// TIA Portal project "RHIKOR Barranquill Agua Renovada_V19" (V19)

(* hardware
DEVICE "S7-1500/ET200MP station_1"  S7-1500 station
   slot 0: "Rail_0"  Rack  6ES7 590-1***0-0AA0
   slot 1: "6ES7 511-1AL03-0AB0"  CPU 1511-1 PN  6ES7 511-1AL03-0AB0  V3.0
      slot 3: "CPU display_1"  6ES7591-1AA00-0AA0
      slot 32768: "PROFINET interface_1"  X1
         slot 32769: "Port_1"  X1 P1
         slot 32770: "Port_2"  X1 P2
      slot 34817: "Virtual CP interface port_1"  Virtual CP interface port  Virtual CP interface port
   slot 2: "PS 25W 24VDC_1"  PS 25W 24VDC  6ES7 505-0KA00-0AB0  V1.1
DEVICE "HMI_1"  KTP900 Basic PN
   slot 0: "HMI_1"  KTP900 Basic PN  6AV2 123-2JB03-0AX0  17.0.0.0
   slot 1: "HMI_RT_1"  KTP900 Basic PN  6AV2 123-2JB03-0AX0  17.0.0.0
   slot 5: "HMI_1.IE_CP_1"  PROFINET Interface  17.0.0.0
      slot 1: "hmixb110d0"  PROFINET Interface
         slot 1: "Port_1"  Port
DEVICE "SCALANCE X005"  SCALANCE X-Station
   slot 0: "SCALANCE X rack"  Rail
   slot 0: "Switch_1"  6GK5 005-0BA00-1AB2  V1.0
DEVICE "ET 200SP station_1"  ET 200SP-Station
   slot 0: "Rack_0"  Rack  6ES5 710-8MAx1
   slot 0: "et200sp"  IM 155-6 PN ST  6ES7 155-6AU02-0BN0  V6.1
   slot 1: "DI 16x24VDC ST_1"  DI 16x24VDC ST  6ES7 131-6BH01-0BA0  V0.0
      slot 1: "DI 16x24VDC ST_1"  DI 16x24VDC ST
   slot 2: "DI 16x24VDC ST_2"  DI 16x24VDC ST  6ES7 131-6BH01-0BA0  V0.0
      slot 1: "DI 16x24VDC ST_2"  DI 16x24VDC ST
   slot 3: "DI 16x24VDC ST_3"  DI 16x24VDC ST  6ES7 131-6BH01-0BA0  V0.0
      slot 1: "DI 16x24VDC ST_3"  DI 16x24VDC ST
   slot 4: "DI 16x24VDC ST_4"  DI 16x24VDC ST  6ES7 131-6BH01-0BA0  V0.0
      slot 1: "DI 16x24VDC ST_4"  DI 16x24VDC ST
   slot 5: "DQ 16x24VDC/0.5A ST_1"  DQ 16x24VDC/0.5A ST  6ES7 132-6BH01-0BA0  V0.0
      slot 1: "DQ 16x24VDC/0.5A ST_1"  DQ 16x24VDC/0.5A ST
   slot 6: "DQ 16x24VDC/0.5A ST_2"  DQ 16x24VDC/0.5A ST  6ES7 132-6BH01-0BA0  V0.0
      slot 1: "DQ 16x24VDC/0.5A ST_2"  DQ 16x24VDC/0.5A ST
   slot 7: "DQ 16x24VDC/0.5A ST_3"  DQ 16x24VDC/0.5A ST  6ES7 132-6BH01-0BA0  V0.0
      slot 1: "DQ 16x24VDC/0.5A ST_3"  DQ 16x24VDC/0.5A ST
   slot 8: "AI 4xU/I 2-wire ST_1"  AI 4xU/I 2-wire ST  6ES7 134-6HD01-0BA1  V2.0
      slot 1: "AI 4xU/I 2-wire ST_1"  AI 4xU/I 2-wire ST
   slot 9: "AI 4xU/I 2-wire ST_2"  AI 4xU/I 2-wire ST  6ES7 134-6HD01-0BA1  V2.0
      slot 1: "AI 4xU/I 2-wire ST_2"  AI 4xU/I 2-wire ST
   slot 10: "AI 4xU/I 2-wire ST_3"  AI 4xU/I 2-wire ST  6ES7 134-6HD01-0BA1  V2.0
      slot 1: "AI 4xU/I 2-wire ST_3"  AI 4xU/I 2-wire ST
   slot 11: "AI 4xU/I 2-wire ST_4"  AI 4xU/I 2-wire ST  6ES7 134-6HD01-0BA1  V2.0
      slot 1: "AI 4xU/I 2-wire ST_4"  AI 4xU/I 2-wire ST
   slot 12: "AI 4xU/I 2-wire ST_5"  AI 4xU/I 2-wire ST  6ES7 134-6HD01-0BA1  V2.0
      slot 1: "AI 4xU/I 2-wire ST_5"  AI 4xU/I 2-wire ST
   slot 13: "AI 4xU/I 2-wire ST_6"  AI 4xU/I 2-wire ST  6ES7 134-6HD01-0BA1  V2.0
      slot 1: "AI 4xU/I 2-wire ST_6"  AI 4xU/I 2-wire ST
   slot 14: "AI 4xU/I 2-wire ST_7"  AI 4xU/I 2-wire ST  6ES7 134-6HD01-0BA1  V2.0
      slot 1: "AI 4xU/I 2-wire ST_7"  AI 4xU/I 2-wire ST
   slot 15: "AQ 4xU/I ST_1"  AQ 4xU/I ST  6ES7 135-6HD00-0BA1  V1.1
      slot 1: "AQ 4xU/I ST_1"  AQ 4xU/I ST
   slot 16: "Server module_1"  Server module  6ES7 193-6PA00-0AA0  V1.1
      slot 1: "Server module_1"  Server module
   slot 127: "BA 2xRJ45"  BA 2xRJ45  6ES7 193-6AR00-0AA0  V0.0
      slot 1: "Port_1"  X1 P1 R  6ES7 193-6AR00-0AA0  V0.0
      slot 2: "Port_2"  X1 P2 R  6ES7 193-6AR00-0AA0  V0.0
*)

// ===== PLC "6ES7 511-1AL03-0AB0"  CPU 1511-1 PN =====

VAR_GLOBAL   // PLC tag table "Default tag table"
   "System_Byte" AT %MB1 : Byte;
   "FirstScan" AT %M1.0 : Bool;
   "DiagStatusUpdate" AT %M1.1 : Bool;
   "AlwaysTRUE" AT %M1.2 : Bool;
   "AlwaysFALSE" AT %M1.3 : Bool;
   "Clock_Byte" AT %MB0 : Byte;
   "Clock_10Hz" AT %M0.0 : Bool;
   "Clock_5Hz" AT %M0.1 : Bool;
   "Clock_2.5Hz" AT %M0.2 : Bool;
   "Clock_2Hz" AT %M0.3 : Bool;
   "Clock_1.25Hz" AT %M0.4 : Bool;
   "Clock_1Hz" AT %M0.5 : Bool;
   "Clock_0.625Hz" AT %M0.6 : Bool;
   "Clock_0.5Hz" AT %M0.7 : Bool;
   "Solito" AT %MW2 : Word;
   "Tag_1" AT %C0 : Counter;
END_VAR

VAR_GLOBAL   // PLC tag table "Entradas"
   "KF1_feedback" AT %I0.0 : Bool;
   "S1_feedback" AT %I0.1 : Bool;
   "BC-08_feedback" AT %I0.2 : Bool;
   "BC-09_feedback" AT %I0.3 : Bool;
   "BC-10_feedback" AT %I0.4 : Bool;
   "BC-11_feedback_protector" AT %I0.5 : Bool;
   "BC-12_feedback" AT %I0.6 : Bool;
   "BC-13_feedback" AT %I0.7 : Bool;
   "BC-14_feedback" AT %I1.0 : Bool;
   "BLW-01_feedback" AT %I1.1 : Bool;
   "UV-01_feedback" AT %I1.2 : Bool;
   "BD-AI-01_feedback" AT %I1.3 : Bool;
   "BD-BIO-01_feedback" AT %I1.4 : Bool;
   "BD-HIP-01_feedback" AT %I1.5 : Bool;
   "BD-HIP-02_feedback" AT %I1.6 : Bool;
   "BD-MBI-01_feedback" AT %I1.7 : Bool;
   "BD-UF-01_feedback" AT %I2.0 : Bool;
   "VM-27-2_feedback" AT %I2.1 : Bool;
   "VM-29_feedback" AT %I2.2 : Bool;
   "VM-31_feedback" AT %I2.3 : Bool;
   "VM-32_feedback" AT %I2.4 : Bool;
   "VM-33_feedback" AT %I2.5 : Bool;
   "VM-34_feedback" AT %I2.6 : Bool;
   "VM-35_feedback" AT %I2.7 : Bool;
   "VM-36_feedback" AT %I3.0 : Bool;
   "VM-39_feedback" AT %I3.1 : Bool;
   "VM-40_feedback" AT %I3.2 : Bool;
   "VM-41_feedback" AT %I3.3 : Bool;
   "VM-42_feedback" AT %I3.4 : Bool;
   "VM-45_feedback" AT %I3.5 : Bool;
   "VM-46_feedback" AT %I3.6 : Bool;
   "VM-47_feedback" AT %I3.7 : Bool;
   "VM-48_feedback" AT %I4.0 : Bool;
   "VM-49_feedback" AT %I4.1 : Bool;
   "VM-50_feedback" AT %I4.2 : Bool;
   "VM-51_feedback" AT %I4.3 : Bool;
   "VM-52_feedback" AT %I4.4 : Bool;
   "VM-53_feedback" AT %I4.5 : Bool;
   "VM-56_feedback" AT %I4.6 : Bool;
   "VM-57_feedback" AT %I4.7 : Bool;
   "VM-58_feedback" AT %I5.0 : Bool;
   "VM-61_feedback" AT %I5.1 : Bool;
   "VM-62_feedback" AT %I5.2 : Bool;
   "VM-63_feedback" AT %I5.3 : Bool;
   "LSH-02_feedback" AT %I5.4 : Bool;
   "LSH-EX1_feedback" AT %I5.5 : Bool;
   "LSL-03_feedback" AT %I5.6 : Bool;
   "LSL-04_feedback" AT %I5.7 : Bool;
   "LSL-05_feedback" AT %I6.0 : Bool;
   "LSL-06_feedback" AT %I6.1 : Bool;
   "LSL-07_feedback" AT %I6.2 : Bool;
   "LSL-08_feedback" AT %I6.3 : Bool;
   "LSL-XX_feedback" AT %I6.4 : Bool;
   "BC-11_feedback_variador" AT %I6.5 : Bool;
   "COT-01_feedback" AT %IW8 : Int;
   "CT-02_feedback" AT %IW10 : Int;
   "FI-06_feedback" AT %IW12 : Int;
   "FI-07_feedback" AT %IW14 : Int;
   "FI-08_feedback" AT %IW16 : Int;
   "FI-09_feedback" AT %IW18 : Int;
   "FI-10_feedback" AT %IW20 : Int;
   "FI-11_feedback" AT %IW22 : Int;
   "ORP-01_feedback" AT %IW24 : Int;
   "ORP-02_feedback" AT %IW26 : Int;
   "PH-04_feedback" AT %IW28 : Int;
   "TRB-02_feedback" AT %IW30 : Int;
   "PT-05_feedback" AT %IW32 : Int;
   "PT-06_feedback" AT %IW34 : Int;
   "PT-07_feedback" AT %IW36 : Int;
   "PT-08_feedback" AT %IW38 : Int;
   "PT-09_feedback" AT %IW40 : Int;
   "PT-10_feedback" AT %IW42 : Int;
   "PT-11_feedback" AT %IW44 : Int;
   "PT-12_feedback" AT %IW46 : Int;
   "PT-13_feedback" AT %IW48 : Int;
   "RAD-04_feedback" AT %IW50 : Int;
   "RAD-05_feedback" AT %IW52 : Int;
   "RAD-06_feedback" AT %IW54 : Int;
END_VAR

VAR_GLOBAL   // PLC tag table "Salidas"
   "BC-08_control" AT %Q0.0 : Bool;
   "BC-09_control" AT %Q0.1 : Bool;
   "BC-10_control" AT %Q0.2 : Bool;
   "BC-11_control" AT %Q0.3 : Bool;
   "BC-12_control" AT %Q0.4 : Bool;
   "BC-13_control" AT %Q0.5 : Bool;
   "BC-14_control" AT %Q0.6 : Bool;
   "BLW-01_control" AT %Q0.7 : Bool;
   "UV-01_control" AT %Q1.0 : Bool;
   "BD-AI-01_control" AT %Q1.1 : Bool;
   "BD-BIO-01_control" AT %Q1.2 : Bool;
   "BD-HIP-01_control" AT %Q1.3 : Bool;
   "BD-HIP-02_control" AT %Q1.4 : Bool;
   "BD-MBI-01_control" AT %Q1.5 : Bool;
   "BD-UF-01_control" AT %Q1.6 : Bool;
   "VM-27-2_control" AT %Q1.7 : Bool;
   "VM-29_control" AT %Q2.0 : Bool;
   "VM-31_control" AT %Q2.1 : Bool;
   "VM-32_control" AT %Q2.2 : Bool;
   "VM-33_control" AT %Q2.3 : Bool;
   "VM-34_control" AT %Q2.4 : Bool;
   "VM-35_control" AT %Q2.5 : Bool;
   "VM-36_control" AT %Q2.6 : Bool;
   "VM-39_control" AT %Q2.7 : Bool;
   "VM-40_control" AT %Q3.0 : Bool;
   "VM-41_control" AT %Q3.1 : Bool;
   "VM-42_control" AT %Q3.2 : Bool;
   "VM-45_control" AT %Q3.3 : Bool;
   "VM-46_control" AT %Q3.4 : Bool;
   "VM-47_control" AT %Q3.5 : Bool;
   "VM-48_control" AT %Q3.6 : Bool;
   "VM-49_control" AT %Q3.7 : Bool;
   "VM-50_control" AT %Q4.0 : Bool;
   "VM-51_control" AT %Q4.1 : Bool;
   "VM-52_control" AT %Q4.2 : Bool;
   "VM-53_control" AT %Q4.3 : Bool;
   "VM-56_control" AT %Q4.4 : Bool;
   "VM-57_control" AT %Q4.5 : Bool;
   "VM-58_control" AT %Q4.6 : Bool;
   "VM-61_control" AT %Q4.7 : Bool;
   "VM-62_control" AT %Q5.0 : Bool;
   "VM-63_control" AT %Q5.1 : Bool;
   "BC-11_frecuencia" AT %QW6 : Int;
END_VAR

TYPE "UDT_VALVULA_NEUMATICA"
   STRUCT
      control : Bool;   // 1=arranque, 0=paro
      feedback : Bool;   // 1=en marcha, 0=detenida
      estado : Int;   // 1=encendida, 2=apagada, 3=alarma
      alarma : Bool;   // 1=alarma activa
      tiempo_alarma : Time := t#3s;   // horas de operación acumuladas
      estado_texto : String;   // ON, OFF, ALARM
   END_STRUCT;
END_TYPE

TYPE "UDT_SENSORES_FLUJO"
   STRUCT
      valor : Int;   // valor actual de flujo
      unidad : String;   // m3/h
      totalizador : DInt;   // contador acumulado
      estado : Int;   // 1=normal, 2=bajo, 3=alto, 4=alarma
      alarma : Bool;   // 1=alarma activa
      estado_texto : String;   // NORMAL, BAJO, ALTO, ALARM
      operacion_alto : Int;   // rango de trabajo alto
      operacion_bajo : Int;   // rango de trabajo bajo
      trabajo_alto : Int;
      trabajo_bajo : Int;
      alarma_bajo : Bool;   // 1=alarma activa
      alarma_alto : Bool;
      flujo : Int;
   END_STRUCT;
END_TYPE

TYPE "UDT_SENSORES_ESPECIALES"
   STRUCT
      valor : Int;   // valor actual
      unidad : String;   // mV, pH, mS/cm, etc.
      operacion_alto : Int;   // rango de trabajo alto
      operacion_bajo : Int;   // rango de trabajo bajo
      estado : Int;   // 1=normal, 2=bajo, 3=alto, 4=alarma
      trabajo_alto : Int;
      trabajo_bajo : Int;
      alarma_bajo : Bool;   // 1=alarma activa
      alarma_alto : Bool;
      estado_texto : String;   // NORMAL, BAJO, ALTO, ALARM
      condicion_alarma : Bool;
      medicion : Int;
   END_STRUCT;
END_TYPE

TYPE "UDT_EQUIPOS_ESPECIALES"
   STRUCT
      control : Bool;   // 1=arranque, 0=paro
      feedback : Bool;   // 1=en marcha, 0=detenida
      proceso : Int;   // proceso asociado (1-10)
      estado : Int;   // 1=encendida, 2=apagada, 3=alarma
      alarma : Bool;   // 1=alarma activa
      horometro : Time;   // horas de operación acumuladas
      estado_texto : String;   // ON, OFF, ALARM
   END_STRUCT;
END_TYPE

TYPE "UDT_BOMBAS"
   STRUCT
      control : Bool;   // 1=arranque, 0=paro
      frecuencia : Int;   // frecuencia variador
      feedback : Bool;   // 1=en marcha, 0=detenida
      tiempo_alarma : Time := T#3s;   // tiempo máximo para arranque
      estado : Int;   // 1=encendida, 2=apagada, 3=alarma
      alarma : Bool;   // 1=alarma activa
      horometro : Time;   // horas de operación acumuladas
      estado_texto : String;
      alarma_variador : Bool;
      valor : Int;
   END_STRUCT;
END_TYPE

TYPE "UDT_BOMBAS_DOSIFICADORAS"
   STRUCT
      control : Bool;   // 1=arranque, 0=paro
      feedback : Bool;   // 1=en marcha, 0=detenida
      nivel_bajo_quimico : Bool;   // 1=nivel bajo en tanque químico
      estado : Int;   // 1=encendida, 2=apagada, 3=alarma
      alarma : Bool;   // 1=alarma activa
      horometro : Time;   // horas de operación acumuladas
      estado_texto : String;
      tiempo_alarma : Time := t#1s;
   END_STRUCT;
END_TYPE

TYPE "UDT_SENSORES_NIVEL"
   STRUCT
      valor : Int;   // valor actual de nivel
      unidad : String;   // m, %
      nivel : Int;   // 1=bajo 2=medio 3=alto
      estado : Int;   // 1=encendida, 2=apagada, 3=alarma
      alarma : Bool;   // 1=alarma activa
      estado_texto : String;   // NORMAL, BAJO, ALTO, ALARM
      alarma_nivel : Bool;
      tiempo_alarma : Time;
      operacion_alto : Int;
      rango_bajo : Int;
      rango_medio_bajo : Int;
      rango_medio_alto : Int;
      rango_alto : Int;
      area_tanque : Int;
      nivel_porcentaje : Int;
      nivel_volumen : Int;
   END_STRUCT;
END_TYPE

TYPE "UDT_SENSORES_PRESION"
   STRUCT
      valor : Int;   // valor actual de presión
      unidad : String := 'BAR';   // bar
      presion : Int;
      estado : Int;   // 1=normal, 2=bajo, 3=alto, 4=alarma
      alarma_alto : Bool;   // 1=alarma activa
      alarma_bajo : Bool;
      estado_texto : String;   // NORMAL, BAJO, ALTO, ALARM
      operacion_alto : Int;   // rango de trabajo alto
      operacion_bajo : Int;   // rango de trabajo bajo
      trabajo_alto : Int;
      trabajo_bajo : Int;
      condicion_alarma : Bool;
   END_STRUCT;
END_TYPE

TYPE "UDT_AUXILIARES"
   STRUCT
      Vigilante_Tension : Bool;
      Paro_Emergencia : Bool;
      tiempo_alarma_valvulas : Time;
   END_STRUCT;
END_TYPE

TYPE "UDT_PRESION_DIFERENCIAL"
   STRUCT
      PresionPT11_PT10 : Int;
   END_STRUCT;
END_TYPE

TYPE "UDT_PRODUCCION_UF"
   STRUCT
      ProcessID : Int := 1;
      ProcessName : String[20] := 'Produccion UF';
      IsActive : Bool;
      IsEnabled : Bool;
      AutoMode : Bool;
      ManualMode : Bool;
      Retrolavado_UF_Active : Bool;
      CIP_UF_Active : Bool;
      CIP_TUF_Active : Bool;
      Refill_UF_Active : Bool;
   END_STRUCT;
END_TYPE

DATA_BLOCK "UDT_Objetos"   // DB1
{ S7_Optimized_Access := 'FALSE' }
VERSION : 0.1
   VAR
      Valvulas : Struct
         "VM-27" : "UDT_VALVULA_NEUMATICA";
         "VM-29" : "UDT_VALVULA_NEUMATICA";
         "VM-31" : "UDT_VALVULA_NEUMATICA";
         "VM-32" : "UDT_VALVULA_NEUMATICA";
         "VM-33" : "UDT_VALVULA_NEUMATICA";
         "VM-34" : "UDT_VALVULA_NEUMATICA";
         "VM-35" : "UDT_VALVULA_NEUMATICA";
         "VM-36" : "UDT_VALVULA_NEUMATICA";
         "VM-39" : "UDT_VALVULA_NEUMATICA";
         "VM-40" : "UDT_VALVULA_NEUMATICA";
         "VM-41" : "UDT_VALVULA_NEUMATICA";
         "VM-42" : "UDT_VALVULA_NEUMATICA";
         "VM-45" : "UDT_VALVULA_NEUMATICA";
         "VM-46" : "UDT_VALVULA_NEUMATICA";
         "VM-47" : "UDT_VALVULA_NEUMATICA";
         "VM-48" : "UDT_VALVULA_NEUMATICA";
         "VM-49" : "UDT_VALVULA_NEUMATICA";
         "VM-50" : "UDT_VALVULA_NEUMATICA";
         "VM-51" : "UDT_VALVULA_NEUMATICA";
         "VM-52" : "UDT_VALVULA_NEUMATICA";
         "VM-53" : "UDT_VALVULA_NEUMATICA";
         "VM-56" : "UDT_VALVULA_NEUMATICA";
         "VM-57" : "UDT_VALVULA_NEUMATICA";
         "VM-58" : "UDT_VALVULA_NEUMATICA";
         "VM-61" : "UDT_VALVULA_NEUMATICA";
         "VM-62" : "UDT_VALVULA_NEUMATICA";
         "VM-63" : "UDT_VALVULA_NEUMATICA";
      END_STRUCT;
      Bombas : Struct
         "BC-08" : "UDT_BOMBAS";
         "BC-09" : "UDT_BOMBAS";
         "BC-10" : "UDT_BOMBAS";
         "BC-11" : "UDT_BOMBAS";
         "BC-12" : "UDT_BOMBAS";
         "BC-13" : "UDT_BOMBAS";
         "BC-14" : "UDT_BOMBAS";
      END_STRUCT;
      Dosificadoras : Struct
         "BD-HIP-01" : "UDT_BOMBAS_DOSIFICADORAS";
         "BD-MBI-01" : "UDT_BOMBAS_DOSIFICADORAS";
         "BD-UF-01" : "UDT_BOMBAS_DOSIFICADORAS";
         "BD-AI-01" : "UDT_BOMBAS_DOSIFICADORAS";
         "BD-BIO-01" : "UDT_BOMBAS_DOSIFICADORAS";
         "BD-HIP-02" : "UDT_BOMBAS_DOSIFICADORAS";
      END_STRUCT;
      Nivel : Struct
         "RAD-04" : "UDT_SENSORES_NIVEL";
         "RAD-05" : "UDT_SENSORES_NIVEL";
         "RAD-06" : "UDT_SENSORES_NIVEL";
         "LSH-EX1" : "UDT_SENSORES_NIVEL";
         "LSL-06" : "UDT_SENSORES_NIVEL";
         "LSH-02" : "UDT_SENSORES_NIVEL";
         "PT-07" : "UDT_SENSORES_NIVEL";
         "PT-12" : "UDT_SENSORES_NIVEL";
         "PT-13" : "UDT_SENSORES_NIVEL";
      END_STRUCT;
      Presion : Struct
         "PT-05" : "UDT_SENSORES_PRESION";
         "PT-06" : "UDT_SENSORES_PRESION";
         "PT-08" : "UDT_SENSORES_PRESION";
         "PT-09" : "UDT_SENSORES_PRESION";
         "PT-10" : "UDT_SENSORES_PRESION";
         "PT-11" : "UDT_SENSORES_PRESION";
      END_STRUCT;
      Flujo : Struct
         "FI-06" : "UDT_SENSORES_FLUJO";
         "FI-07" : "UDT_SENSORES_FLUJO";
         "FI-08" : "UDT_SENSORES_FLUJO";
         "FI-09" : "UDT_SENSORES_FLUJO";
         "FI-10" : "UDT_SENSORES_FLUJO";
         "FI-11" : "UDT_SENSORES_FLUJO";
      END_STRUCT;
      Sensores_Especiales : Struct
         "TRB-02" : "UDT_SENSORES_ESPECIALES";
         "ORP-01" : "UDT_SENSORES_ESPECIALES";
         "ORP-02" : "UDT_SENSORES_ESPECIALES";
         "PH-04" : "UDT_SENSORES_ESPECIALES";
         "CT-02" : "UDT_SENSORES_ESPECIALES";
         "COT-01" : "UDT_SENSORES_ESPECIALES";
      END_STRUCT;
      Equipos_Especiales : Struct
         "BLW-01" : "UDT_EQUIPOS_ESPECIALES";
         "UV-01" : "UDT_EQUIPOS_ESPECIALES";
      END_STRUCT;
      Auxiliares : Struct
         AuxiliaresGenerales : "UDT_AUXILIARES";
         PresionDiferencial : "UDT_PRESION_DIFERENCIAL";
      END_STRUCT;
      PresionDiferencial : "UDT_AUXILIARES";
      AlarmasTotales : Struct
         AlarmasValvulas1 : Int;
         AlarmasValvulas2 : Int;
         AlarmasPresion : Int;
         AlarmasEspeciales : Int;
         AlarmasDosificadoras : Int;
         AlarmasBombas : Int;
         AlarmasFlujo : Int;
         AlarmasTanques : Int;
      END_STRUCT;
      ProcesoUF : "UDT_PRODUCCION_UF";
   END_VAR
BEGIN
   Bombas."BC-11".frecuencia := 60;
   Sensores_Especiales."COT-01".operacion_alto := 0;
   Sensores_Especiales."COT-01".operacion_bajo := 100;
   Sensores_Especiales."COT-01".trabajo_alto := 4;
   Sensores_Especiales."COT-01".trabajo_bajo := 5;
   Sensores_Especiales."CT-02".operacion_bajo := 0;
   Sensores_Especiales."CT-02".operacion_alto := 2000;
   Sensores_Especiales."CT-02".trabajo_alto := 190;
   Sensores_Especiales."CT-02".trabajo_bajo := 130;
   Sensores_Especiales."ORP-01".operacion_alto := 2000;
   Sensores_Especiales."ORP-01".operacion_bajo := -2000;
   Sensores_Especiales."ORP-02".operacion_alto := 2000;
   Sensores_Especiales."ORP-02".operacion_bajo := -2000;
   Sensores_Especiales."ORP-01".trabajo_alto := 600;
   Sensores_Especiales."ORP-01".trabajo_bajo := 600;
   Sensores_Especiales."ORP-02".trabajo_alto := 600;
   Sensores_Especiales."ORP-02".trabajo_bajo := 600;
   Sensores_Especiales."PH-04".operacion_alto := 14;
   Sensores_Especiales."PH-04".operacion_bajo := 0;
   Sensores_Especiales."TRB-02".operacion_alto := 2000;
   Sensores_Especiales."TRB-02".operacion_bajo := 0;
   Sensores_Especiales."TRB-02".trabajo_alto := 1100;
   Sensores_Especiales."TRB-02".trabajo_bajo := 900;
   Flujo."FI-06".operacion_alto := 200;
   Flujo."FI-06".operacion_bajo := 0;
   Flujo."FI-06".trabajo_alto := 125;
   Flujo."FI-06".trabajo_bajo := 115;
   Flujo."FI-07".operacion_alto := 200;
   Flujo."FI-07".operacion_bajo := 0;
   Flujo."FI-07".trabajo_alto := 125;
   Flujo."FI-07".trabajo_bajo := 115;
   Flujo."FI-08".operacion_alto := 200;
   Flujo."FI-08".operacion_bajo := 0;
   Flujo."FI-08".trabajo_alto := 125;
   Flujo."FI-08".trabajo_bajo := 115;
   Flujo."FI-09".operacion_alto := 150;
   Flujo."FI-09".operacion_bajo := 0;
   Flujo."FI-09".trabajo_alto := 85;
   Flujo."FI-09".trabajo_bajo := 83;
   Flujo."FI-10".operacion_alto := 100;
   Flujo."FI-10".operacion_bajo := 0;
   Flujo."FI-10".trabajo_alto := 37;
   Flujo."FI-10".trabajo_bajo := 35;
   Nivel."RAD-04".operacion_alto := 80;
   Nivel."RAD-04".rango_bajo := 10;
   Nivel."RAD-04".rango_medio_bajo := 15;
   Nivel."RAD-04".rango_medio_alto := 35;
   Nivel."RAD-04".rango_alto := 40;
   Nivel."RAD-05".operacion_alto := 80;
   Nivel."RAD-05".rango_bajo := 10;
   Nivel."RAD-05".rango_medio_bajo := 15;
   Nivel."RAD-05".rango_medio_alto := 35;
   Nivel."RAD-05".rango_alto := 40;
   Nivel."RAD-06".operacion_alto := 80;
   Nivel."RAD-06".rango_bajo := 10;
   Nivel."RAD-06".rango_medio_bajo := 15;
   Nivel."RAD-06".rango_medio_alto := 35;
   Nivel."RAD-06".rango_alto := 40;
   Presion."PT-05".operacion_alto := 40;
   Presion."PT-05".operacion_bajo := 0;
   Presion."PT-05".trabajo_alto := 35;
   Presion."PT-05".trabajo_bajo := 15;
   Presion."PT-06".operacion_alto := 40;
   Presion."PT-06".operacion_bajo := 0;
   Presion."PT-06".trabajo_alto := 35;
   Presion."PT-06".trabajo_bajo := 15;
   Presion."PT-08".operacion_alto := 40;
   Presion."PT-08".operacion_bajo := 0;
   Presion."PT-08".trabajo_alto := 35;
   Presion."PT-08".trabajo_bajo := 15;
   Presion."PT-09".operacion_alto := 200;
   Presion."PT-09".operacion_bajo := 0;
   Presion."PT-09".trabajo_alto := 77;
   Presion."PT-09".trabajo_bajo := 63;
   Presion."PT-10".operacion_alto := 200;
   Presion."PT-10".operacion_bajo := 0;
   Presion."PT-10".trabajo_alto := 20;
   Presion."PT-10".trabajo_bajo := 0;
   Presion."PT-11".operacion_alto := 200;
   Presion."PT-11".operacion_bajo := 0;
   Presion."PT-11".trabajo_alto := 77;
   Presion."PT-11".trabajo_bajo := 63;
   Nivel."PT-07".operacion_alto := 10;
   Nivel."PT-07".rango_bajo := 1;
   Nivel."PT-07".rango_medio_bajo := 3;
   Nivel."PT-07".rango_medio_alto := 8;
   Nivel."PT-07".rango_alto := 13;
   Nivel."PT-12".operacion_alto := 10;
   Nivel."PT-12".rango_bajo := 1;
   Nivel."PT-12".rango_medio_bajo := 3;
   Nivel."PT-12".rango_medio_alto := 8;
   Nivel."PT-12".rango_alto := 13;
   Nivel."PT-13".operacion_alto := 10;
   Nivel."PT-13".rango_bajo := 1;
   Nivel."PT-13".rango_medio_bajo := 3;
   Nivel."PT-13".rango_medio_alto := 12;
   Nivel."PT-13".rango_alto := 14;
   Flujo."FI-11".operacion_alto := 100;
   Flujo."FI-11".operacion_bajo := 0;
   Flujo."FI-11".trabajo_alto := 37;
   Flujo."FI-11".trabajo_bajo := 35;
   Nivel."RAD-04".area_tanque := 1;
   Nivel."RAD-05".area_tanque := 1;
   Nivel."RAD-06".area_tanque := 1;
   Nivel."PT-07".area_tanque := 1;
   Nivel."PT-12".area_tanque := 1;
   Nivel."PT-13".area_tanque := 1;
END_DATA_BLOCK

DATA_BLOCK "Default_SupervisionDB"   // DB5
{ S7_Optimized_Access := 'TRUE' }
VERSION : 0.1
// stored: InstanceOfName Default_SupervisionFB
"Default_SupervisionFB"
BEGIN
END_DATA_BLOCK

// folder: Alarmas_Totales/Bloques_Datos

DATA_BLOCK "GrupoErroresValvulas_DB"   // DB2
{ S7_Optimized_Access := 'TRUE' }
VERSION : 0.1
// stored: InstanceOfName GrupoErroresValvulas
"GrupoErroresValvulas"
BEGIN
END_DATA_BLOCK

// folder: Estados/Bloques_Datos

DATA_BLOCK "InstanciasValvulas_DB"   // DB3
{ S7_Optimized_Access := 'TRUE' }
VERSION : 0.1
// stored: InstanceOfName InstanciasValvulas
"InstanciasValvulas"
BEGIN
END_DATA_BLOCK

// folder: Procesos

DATA_BLOCK "AutomaticoUF_DB"   // DB4
{ S7_Optimized_Access := 'TRUE' }
VERSION : 0.1
// stored: InstanceOfName AutomaticoUF
"AutomaticoUF"
BEGIN
END_DATA_BLOCK

// folder: (top level)

FUNCTION_BLOCK "Default_SupervisionFB"   // FB18, ProDiag
{ S7_Optimized_Access := 'TRUE' }
   VAR
      PC_Flags : PC_Flags_V2;
      State : SV_FB_State_V2;
      "UDT_Objetos.Valvulas.VM-63.control_O_1" : SV_State_V2;
      Glob_Err_C1 : Diag_Alarm_2;
   END_VAR
   VAR_TEMP
      t_TempSvStateUDT : SV_State_V2;
      t_TempAlarmInstance : <type 200004f>;
      t_TempAsocValue1 : Variant;
      t_TempAsocValue2 : Variant;
      t_TempAsocValue3 : Variant;
   END_VAR
BEGIN
END_FUNCTION_BLOCK

ORGANIZATION_BLOCK "Main"   // OB1, LAD, ProgramCycle
TITLE = "Main Program Sweep (Cycle)"
{ S7_Optimized_Access := 'TRUE' }
VERSION : 0.1
   VAR_INPUT
      Initial_Call : Bool;   // Initial call of this OB
      Remanence : Bool;   // =True, if remanent data are available
   END_VAR
BEGIN
END_ORGANIZATION_BLOCK

ORGANIZATION_BLOCK "ProDiagOB"   // OB250, ProDiag_OB, ProgramCycle
TITLE = "Main Program Sweep (Cycle)"
{ S7_Optimized_Access := 'TRUE' }
VERSION : 0.1
   VAR_INPUT
      Initial_Call : Bool;   // Initial call of this OB
      Remanence : Bool;   // =True, if remanent data are available
   END_VAR
BEGIN

REGION Network 1
   CALL "Default_SupervisionFB", "Default_SupervisionDB";
END_REGION
END_ORGANIZATION_BLOCK

// folder: Alarmas_Totales

FUNCTION_BLOCK "AlarmasValvulas"   // FB1, LAD
{ S7_Optimized_Access := 'TRUE' }
VERSION : 0.1
   VAR_OUTPUT
      AlarmaStruct : Bool;
   END_VAR
   VAR_IN_OUT
      Instancia_Valvula : "UDT_VALVULA_NEUMATICA";
   END_VAR
   VAR
      TemporizadorAlarma : TOF_TIME;
      Auxiliares : Struct
         A1 : Bool;
         A2 : Bool;
         A3 : Bool;
         A4 : Bool;
         A5 : Bool;
         A6 : Bool;
         A7 : Bool;
      END_STRUCT;
   END_VAR
   VAR_TEMP   // added for the SCL form of the ladder/FBD networks
      _w1 : Bool;
      _w2 : Bool;
      _w3 : Bool;
      _w4 : Bool;
      _w5 : Bool;
   END_VAR
BEGIN

REGION Network 1
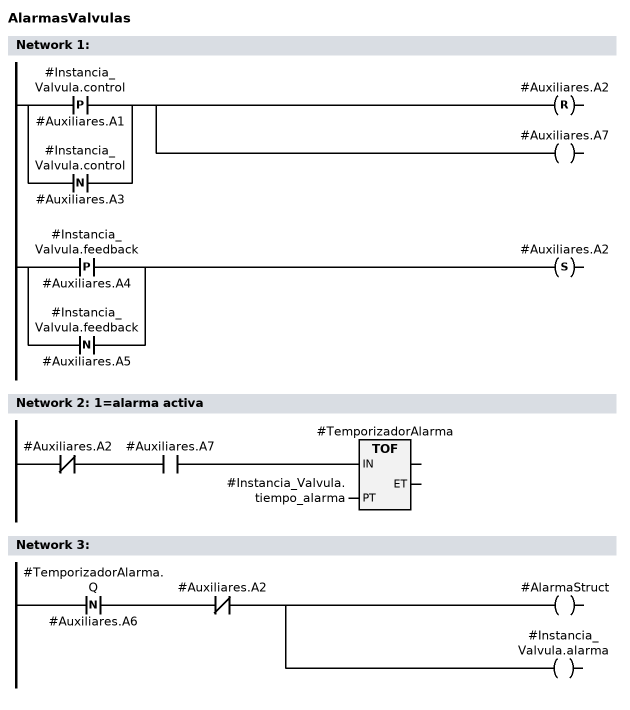
   RUNG wire#powerrail
      P_Contact(operand := #Instancia_Valvula.control, bit := #Auxiliares.A1)
      wire#w1
      R_Coil( #Auxiliares.A2 )
   END_RUNG
   RUNG wire#powerrail
      N_Contact(operand := #Instancia_Valvula.control, bit := #Auxiliares.A3)
   END_RUNG wire#w1
   RUNG wire#w1
      Coil( #Auxiliares.A7 )
   END_RUNG
   RUNG wire#powerrail
      P_Contact(operand := #Instancia_Valvula.feedback, bit := #Auxiliares.A4)
      wire#w2
      S_Coil( #Auxiliares.A2 )
   END_RUNG
   RUNG wire#powerrail
      N_Contact(operand := #Instancia_Valvula.feedback, bit := #Auxiliares.A5)
   END_RUNG wire#w2
   // the same network as SCL:
   #_w1 := #Instancia_Valvula.control AND NOT #Auxiliares.A1;   // rising edge of #Instancia_Valvula.control
   #Auxiliares.A1 := #Instancia_Valvula.control;
   #_w2 := NOT #Instancia_Valvula.control AND #Auxiliares.A3;   // falling edge of #Instancia_Valvula.control
   #Auxiliares.A3 := #Instancia_Valvula.control;
   #_w3 := #_w1 OR #_w2;
   IF #_w3 THEN #Auxiliares.A2 := FALSE; END_IF;
   #Auxiliares.A7 := #_w3;
   #_w4 := #Instancia_Valvula.feedback AND NOT #Auxiliares.A4;   // rising edge of #Instancia_Valvula.feedback
   #Auxiliares.A4 := #Instancia_Valvula.feedback;
   #_w5 := NOT #Instancia_Valvula.feedback AND #Auxiliares.A5;   // falling edge of #Instancia_Valvula.feedback
   #Auxiliares.A5 := #Instancia_Valvula.feedback;
   IF #_w4 OR #_w5 THEN #Auxiliares.A2 := TRUE; END_IF;
END_REGION

REGION Network 2: 1=alarma activa
   #TemporizadorAlarma(IN := NOT #Auxiliares.A2 AND #Auxiliares.A7, PT := #Instancia_Valvula.tiempo_alarma);   // TOF
END_REGION

REGION Network 3
   RUNG wire#powerrail
      N_Contact(operand := #TemporizadorAlarma.Q, bit := #Auxiliares.A6)
      I_Contact( #Auxiliares.A2 )
      wire#w1
      Coil( #AlarmaStruct )
   END_RUNG
   RUNG wire#w1
      Coil( #Instancia_Valvula.alarma )
   END_RUNG
   // the same network as SCL:
   #_w1 := NOT #TemporizadorAlarma.Q AND #Auxiliares.A6;   // falling edge of #TemporizadorAlarma.Q
   #Auxiliares.A6 := #TemporizadorAlarma.Q;
   #AlarmaStruct := #_w1 AND NOT #Auxiliares.A2;
   #Instancia_Valvula.alarma := #AlarmaStruct;
END_REGION
END_FUNCTION_BLOCK

FUNCTION_BLOCK "GrupoErroresValvulas"   // FB2, SCL
{ S7_Optimized_Access := 'TRUE' }
VERSION : 0.1
   VAR
      VM27 : "AlarmasValvulas";
      VM29 : "AlarmasValvulas";
      VM31 : "AlarmasValvulas";
      VM32 : "AlarmasValvulas";
      VM33 : "AlarmasValvulas";
      VM34 : "AlarmasValvulas";
      VM35 : "AlarmasValvulas";
      VM36 : "AlarmasValvulas";
      VM39 : "AlarmasValvulas";
      VM40 : "AlarmasValvulas";
      VM41 : "AlarmasValvulas";
      VM42 : "AlarmasValvulas";
      VM45 : "AlarmasValvulas";
      VM46 : "AlarmasValvulas";
      VM47 : "AlarmasValvulas";
      VM48 : "AlarmasValvulas";
      VM49 : "AlarmasValvulas";
      VM50 : "AlarmasValvulas";
      VM51 : "AlarmasValvulas";
      VM52 : "AlarmasValvulas";
      VM53 : "AlarmasValvulas";
      VM56 : "AlarmasValvulas";
      VM57 : "AlarmasValvulas";
      VM58 : "AlarmasValvulas";
      VM61 : "AlarmasValvulas";
      VM62 : "AlarmasValvulas";
      VM63 : "AlarmasValvulas";
      BC08 : "AlarmasBombas";
      BC09 : "AlarmasBombas";
      BC10 : "AlarmasBombas";
      BC11 : "AlarmasBombas";
      BC12 : "AlarmasBombas";
      BC13 : "AlarmasBombas";
      BC14 : "AlarmasBombas";
      BDAI01 : "AlarmasDosificadoras";
      BDBIO01 : "AlarmasDosificadoras";
      BDHIP01 : "AlarmasDosificadoras";
      BDHIP02 : "AlarmasDosificadoras";
      BDMBI01 : "AlarmasDosificadoras";
      BDUF01 : "AlarmasDosificadoras";
      COT01 : "AlarmasSensoresEspeciales";
      CT02 : "AlarmasSensoresEspeciales";
      ORP01 : "AlarmasSensoresEspeciales";
      ORP02 : "AlarmasSensoresEspeciales";
      PH04 : "AlarmasSensoresEspeciales";
      TRB02 : "AlarmasSensoresEspeciales";
      PT05 : "AlarmasPresioOsmosis";
      PT06 : "AlarmasPresioOsmosis";
      PT08 : "AlarmasPresioOsmosis";
      PT09 : "AlarmasPresioOsmosis";
      PT10PT11 : "AlarmaPresionDiferencial";
      FI06 : "AlarmasFlujo";
      FI07 : "AlarmasFlujo";
      FI08 : "AlarmasFlujo";
      FI09 : "AlarmasFlujo";
   END_VAR
BEGIN
   //VALVULAS
   #VM27(AlarmaStruct=>"UDT_Objetos".AlarmasTotales.AlarmasValvulas1.%X0,
         Instancia_Valvula:="UDT_Objetos".Valvulas."VM-27");
   #VM29(AlarmaStruct => "UDT_Objetos".AlarmasTotales.AlarmasValvulas1.%X1,
         Instancia_Valvula := "UDT_Objetos".Valvulas."VM-29");
   #VM31(AlarmaStruct => "UDT_Objetos".AlarmasTotales.AlarmasValvulas1.%X2,
         Instancia_Valvula := "UDT_Objetos".Valvulas."VM-31");
   #VM32(AlarmaStruct => "UDT_Objetos".AlarmasTotales.AlarmasValvulas1.%X3,
         Instancia_Valvula := "UDT_Objetos".Valvulas."VM-32");
   #VM33(AlarmaStruct => "UDT_Objetos".AlarmasTotales.AlarmasValvulas1.%X4,
         Instancia_Valvula := "UDT_Objetos".Valvulas."VM-33");
   #VM34(AlarmaStruct => "UDT_Objetos".AlarmasTotales.AlarmasValvulas1.%X5,
         Instancia_Valvula := "UDT_Objetos".Valvulas."VM-34");
   #VM35(AlarmaStruct => "UDT_Objetos".AlarmasTotales.AlarmasValvulas1.%X6,
         Instancia_Valvula := "UDT_Objetos".Valvulas."VM-35");
   #VM36(AlarmaStruct => "UDT_Objetos".AlarmasTotales.AlarmasValvulas1.%X7,
         Instancia_Valvula := "UDT_Objetos".Valvulas."VM-36");
   #VM39(AlarmaStruct => "UDT_Objetos".AlarmasTotales.AlarmasValvulas1.%X8,
         Instancia_Valvula := "UDT_Objetos".Valvulas."VM-39");
   #VM40(AlarmaStruct => "UDT_Objetos".AlarmasTotales.AlarmasValvulas1.%X9,
         Instancia_Valvula := "UDT_Objetos".Valvulas."VM-40");
   #VM41(AlarmaStruct => "UDT_Objetos".AlarmasTotales.AlarmasValvulas1.%X10,
         Instancia_Valvula := "UDT_Objetos".Valvulas."VM-41");
   #VM42(AlarmaStruct => "UDT_Objetos".AlarmasTotales.AlarmasValvulas1.%X11,
         Instancia_Valvula := "UDT_Objetos".Valvulas."VM-42");
   #VM45(AlarmaStruct => "UDT_Objetos".AlarmasTotales.AlarmasValvulas1.%X12,
         Instancia_Valvula := "UDT_Objetos".Valvulas."VM-45");
   #VM46(AlarmaStruct => "UDT_Objetos".AlarmasTotales.AlarmasValvulas1.%X13,
         Instancia_Valvula := "UDT_Objetos".Valvulas."VM-46");
   #VM47(AlarmaStruct => "UDT_Objetos".AlarmasTotales.AlarmasValvulas1.%X14,
         Instancia_Valvula := "UDT_Objetos".Valvulas."VM-47");
   #VM48(AlarmaStruct => "UDT_Objetos".AlarmasTotales.AlarmasValvulas1.%X15,
         Instancia_Valvula := "UDT_Objetos".Valvulas."VM-48");
   #VM49(AlarmaStruct => "UDT_Objetos".AlarmasTotales.AlarmasValvulas1.%X0,
         Instancia_Valvula := "UDT_Objetos".Valvulas."VM-49");
   #VM50(AlarmaStruct => "UDT_Objetos".AlarmasTotales.AlarmasValvulas2.%X1,
         Instancia_Valvula := "UDT_Objetos".Valvulas."VM-50");
   #VM51(AlarmaStruct => "UDT_Objetos".AlarmasTotales.AlarmasValvulas2.%X2,
         Instancia_Valvula := "UDT_Objetos".Valvulas."VM-51");
   #VM52(AlarmaStruct => "UDT_Objetos".AlarmasTotales.AlarmasValvulas2.%X3,
         Instancia_Valvula := "UDT_Objetos".Valvulas."VM-52");
   #VM53(AlarmaStruct => "UDT_Objetos".AlarmasTotales.AlarmasValvulas2.%X4,
         Instancia_Valvula := "UDT_Objetos".Valvulas."VM-53");
   #VM56(AlarmaStruct => "UDT_Objetos".AlarmasTotales.AlarmasValvulas2.%X5,
         Instancia_Valvula := "UDT_Objetos".Valvulas."VM-56");
   #VM57(AlarmaStruct => "UDT_Objetos".AlarmasTotales.AlarmasValvulas2.%X6,
         Instancia_Valvula := "UDT_Objetos".Valvulas."VM-57");
   #VM58(AlarmaStruct => "UDT_Objetos".AlarmasTotales.AlarmasValvulas2.%X7,
         Instancia_Valvula := "UDT_Objetos".Valvulas."VM-58");
   #VM61(AlarmaStruct => "UDT_Objetos".AlarmasTotales.AlarmasValvulas2.%X8,
         Instancia_Valvula := "UDT_Objetos".Valvulas."VM-61");
   #VM62(AlarmaStruct => "UDT_Objetos".AlarmasTotales.AlarmasValvulas2.%X9,
         Instancia_Valvula := "UDT_Objetos".Valvulas."VM-62");
   #VM63(AlarmaStruct => "UDT_Objetos".AlarmasTotales.AlarmasValvulas2.%X10,
         Instancia_Valvula := "UDT_Objetos".Valvulas."VM-63");


   //BOMBAS
   #BC08(AlarmaStruct=>"UDT_Objetos".AlarmasTotales.AlarmasBombas.%X0,
         Instancia_Valvula:="UDT_Objetos".Bombas."BC-08");
   #BC09(AlarmaStruct => "UDT_Objetos".AlarmasTotales.AlarmasBombas.%X1,
         Instancia_Valvula := "UDT_Objetos".Bombas."BC-09");
   #BC10(AlarmaStruct => "UDT_Objetos".AlarmasTotales.AlarmasBombas.%X2,
         Instancia_Valvula := "UDT_Objetos".Bombas."BC-10");
   #BC11(AlarmaStruct => "UDT_Objetos".AlarmasTotales.AlarmasBombas.%X3,
         Instancia_Valvula := "UDT_Objetos".Bombas."BC-11");
   #BC12(AlarmaStruct => "UDT_Objetos".AlarmasTotales.AlarmasBombas.%X4,
         Instancia_Valvula := "UDT_Objetos".Bombas."BC-12");
   #BC13(AlarmaStruct => "UDT_Objetos".AlarmasTotales.AlarmasBombas.%X5,
         Instancia_Valvula := "UDT_Objetos".Bombas."BC-13");
   #BC14(AlarmaStruct=>"UDT_Objetos".AlarmasTotales.AlarmasBombas.%X6,
         Instancia_Valvula:="UDT_Objetos".Bombas."BC-14");


   //BOMBAS DOSIFICADORAS
   #BDAI01(AlarmaStruct=>"UDT_Objetos".AlarmasTotales.AlarmasDosificadoras.%X0,
           Instancia_Valvula:="UDT_Objetos".Dosificadoras."BD-AI-01");
   #BDBIO01(AlarmaStruct => "UDT_Objetos".AlarmasTotales.AlarmasDosificadoras.%X1,
            Instancia_Valvula := "UDT_Objetos".Dosificadoras."BD-BIO-01");
   #BDHIP01(AlarmaStruct => "UDT_Objetos".AlarmasTotales.AlarmasDosificadoras.%X2,
            Instancia_Valvula := "UDT_Objetos".Dosificadoras."BD-HIP-01");
   #BDHIP02(AlarmaStruct => "UDT_Objetos".AlarmasTotales.AlarmasDosificadoras.%X3,
            Instancia_Valvula := "UDT_Objetos".Dosificadoras."BD-HIP-02");
   #BDMBI01(AlarmaStruct => "UDT_Objetos".AlarmasTotales.AlarmasDosificadoras.%X4,
            Instancia_Valvula := "UDT_Objetos".Dosificadoras."BD-MBI-01");
   #BDUF01(AlarmaStruct => "UDT_Objetos".AlarmasTotales.AlarmasDosificadoras.%X5,
           Instancia_Valvula := "UDT_Objetos".Dosificadoras."BD-UF-01");

   //Sensores especiales
   #COT01(AlarmaStruct_Alto => "UDT_Objetos".AlarmasTotales.AlarmasEspeciales.%X1,
          FallaGeneral=>"UDT_Objetos".AlarmasTotales.AlarmasEspeciales.%X0,
          Sensor := "UDT_Objetos".Sensores_Especiales."COT-01");
   #CT02(AlarmaStruct_Alto=>"UDT_Objetos".AlarmasTotales.AlarmasEspeciales.%X4,
         AlarmaStruct_Bajo=>"UDT_Objetos".AlarmasTotales.AlarmasEspeciales.%X5,
         FallaGeneral=>"UDT_Objetos".AlarmasTotales.AlarmasEspeciales.%X3,
         Sensor := "UDT_Objetos".Sensores_Especiales."CT-02");

   #ORP01(AlarmaStruct_Alto => "UDT_Objetos".AlarmasTotales.AlarmasEspeciales.%X7,
          FallaGeneral=>"UDT_Objetos".AlarmasTotales.AlarmasEspeciales.%X6,
          Sensor := "UDT_Objetos".Sensores_Especiales."ORP-01");

   #ORP02(AlarmaStruct_Alto => "UDT_Objetos".AlarmasTotales.AlarmasEspeciales.%X9,
          AlarmaStruct_Bajo => "UDT_Objetos".AlarmasTotales.AlarmasEspeciales.%X10,
          FallaGeneral=>"UDT_Objetos".AlarmasTotales.AlarmasEspeciales.%X8,
          Sensor := "UDT_Objetos".Sensores_Especiales."ORP-02");

   #PH04(FallaGeneral => "UDT_Objetos".AlarmasTotales.AlarmasEspeciales.%X12,
         Sensor := "UDT_Objetos".Sensores_Especiales."PH-04");

   #TRB02(AlarmaStruct_Alto => "UDT_Objetos".AlarmasTotales.AlarmasEspeciales.%X14,
          AlarmaStruct_Bajo => "UDT_Objetos".AlarmasTotales.AlarmasEspeciales.%X15,
          FallaGeneral=>"UDT_Objetos".AlarmasTotales.AlarmasEspeciales.%X13,
          Sensor := "UDT_Objetos".Sensores_Especiales."TRB-02");

   //Sensores de flujo directos
   #FI06(Sensor := "UDT_Objetos".Flujo."FI-06",
         AlarmaStruct_Alto => "UDT_Objetos".AlarmasTotales.AlarmasFlujo.%X0,
         AlarmaStruct_Bajo=>"UDT_Objetos".AlarmasTotales.AlarmasFlujo.%X1);
   #FI07(Sensor := "UDT_Objetos".Flujo."FI-07",
         AlarmaStruct_Alto => "UDT_Objetos".AlarmasTotales.AlarmasFlujo.%X2,
         AlarmaStruct_Bajo => "UDT_Objetos".AlarmasTotales.AlarmasFlujo.%X3);
   #FI08(Sensor := "UDT_Objetos".Flujo."FI-08",
         AlarmaStruct_Alto => "UDT_Objetos".AlarmasTotales.AlarmasFlujo.%X4,
         AlarmaStruct_Bajo => "UDT_Objetos".AlarmasTotales.AlarmasFlujo.%X5);
   #FI09(Sensor := "UDT_Objetos".Flujo."FI-09",
         AlarmaStruct_Alto => "UDT_Objetos".AlarmasTotales.AlarmasFlujo.%X6,
         AlarmaStruct_Bajo => "UDT_Objetos".AlarmasTotales.AlarmasFlujo.%X7);

   //Sensores de flujo indirectos
   //FI10





   //Sensores de presion
   #PT05(AlarmaStruct_Alto => "UDT_Objetos".AlarmasTotales.AlarmasPresion.%X1,
         AlarmaStruct_Bajo => "UDT_Objetos".AlarmasTotales.AlarmasPresion.%X0,
         SensorPresion := "UDT_Objetos".Presion."PT-05");
   #PT06(AlarmaStruct_Alto => "UDT_Objetos".AlarmasTotales.AlarmasPresion.%X3,
         AlarmaStruct_Bajo => "UDT_Objetos".AlarmasTotales.AlarmasPresion.%X2,
         SensorPresion := "UDT_Objetos".Presion."PT-06");
   #PT08(AlarmaStruct_Bajo => "UDT_Objetos".AlarmasTotales.AlarmasPresion.%X4,
         SensorPresion := "UDT_Objetos".Presion."PT-08");
   #PT09(AlarmaStruct_Alto => "UDT_Objetos".AlarmasTotales.AlarmasPresion.%X6,
         AlarmaStruct_Bajo => "UDT_Objetos".AlarmasTotales.AlarmasPresion.%X5,
          SensorPresion := "UDT_Objetos".Presion."PT-09");
   #PT10PT11(PresionALcanzada=>"UDT_Objetos".AlarmasTotales.AlarmasPresion.%X7,
              SensorPT10:="UDT_Objetos".Presion."PT-10",
              SensorPT11:="UDT_Objetos".Presion."PT-11",
              Diferencial:="UDT_Objetos".Auxiliares.PresionDiferencial);
   //Sensores de presion para nivel
END_FUNCTION_BLOCK

FUNCTION_BLOCK "AlarmasBombas"   // FB5, LAD
{ S7_Optimized_Access := 'TRUE' }
VERSION : 0.1
   VAR_OUTPUT
      AlarmaStruct : Bool;
   END_VAR
   VAR_IN_OUT
      Instancia_Valvula : "UDT_BOMBAS";
   END_VAR
   VAR
      TemporizadorAlarma : TP_TIME;
      Auxiliares : Struct
         A1 : Bool;
         A2 : Bool;
         A3 : Bool;
         A4 : Bool;
         A5 : Bool;
         A6 : Bool;
         A7 : Bool;
      END_STRUCT;
   END_VAR
   VAR_TEMP   // added for the SCL form of the ladder/FBD networks
      _w1 : Bool;
      _w2 : Bool;
      _w3 : Bool;
      _w4 : Bool;
      _w5 : Bool;
   END_VAR
BEGIN

REGION Network 1
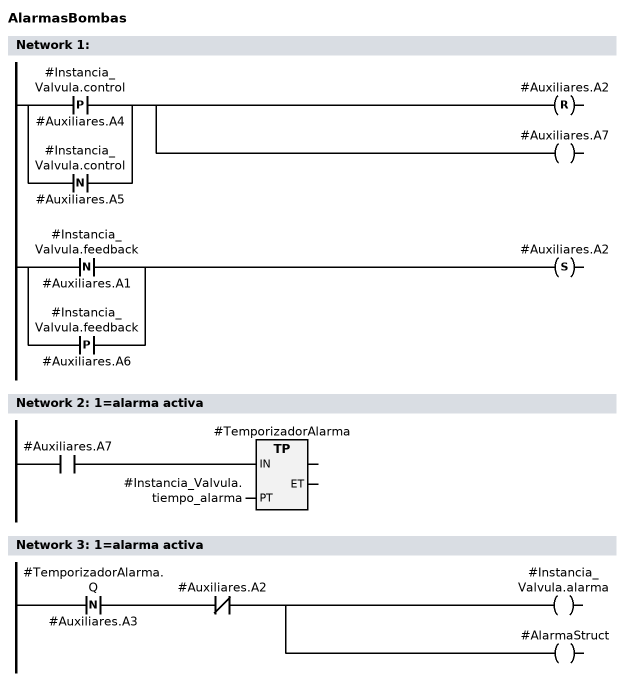
   RUNG wire#powerrail
      P_Contact(operand := #Instancia_Valvula.control, bit := #Auxiliares.A4)
      wire#w1
      R_Coil( #Auxiliares.A2 )
   END_RUNG
   RUNG wire#powerrail
      N_Contact(operand := #Instancia_Valvula.control, bit := #Auxiliares.A5)
   END_RUNG wire#w1
   RUNG wire#w1
      Coil( #Auxiliares.A7 )
   END_RUNG
   RUNG wire#powerrail
      N_Contact(operand := #Instancia_Valvula.feedback, bit := #Auxiliares.A1)
      wire#w2
      S_Coil( #Auxiliares.A2 )
   END_RUNG
   RUNG wire#powerrail
      P_Contact(operand := #Instancia_Valvula.feedback, bit := #Auxiliares.A6)
   END_RUNG wire#w2
   // the same network as SCL:
   #_w1 := #Instancia_Valvula.control AND NOT #Auxiliares.A4;   // rising edge of #Instancia_Valvula.control
   #Auxiliares.A4 := #Instancia_Valvula.control;
   #_w2 := NOT #Instancia_Valvula.control AND #Auxiliares.A5;   // falling edge of #Instancia_Valvula.control
   #Auxiliares.A5 := #Instancia_Valvula.control;
   #_w3 := #_w1 OR #_w2;
   IF #_w3 THEN #Auxiliares.A2 := FALSE; END_IF;
   #Auxiliares.A7 := #_w3;
   #_w4 := NOT #Instancia_Valvula.feedback AND #Auxiliares.A1;   // falling edge of #Instancia_Valvula.feedback
   #Auxiliares.A1 := #Instancia_Valvula.feedback;
   #_w5 := #Instancia_Valvula.feedback AND NOT #Auxiliares.A6;   // rising edge of #Instancia_Valvula.feedback
   #Auxiliares.A6 := #Instancia_Valvula.feedback;
   IF #_w4 OR #_w5 THEN #Auxiliares.A2 := TRUE; END_IF;
END_REGION

REGION Network 2: 1=alarma activa
   #TemporizadorAlarma(IN := #Auxiliares.A7, PT := #Instancia_Valvula.tiempo_alarma);   // TP
END_REGION

REGION Network 3: 1=alarma activa
   RUNG wire#powerrail
      N_Contact(operand := #TemporizadorAlarma.Q, bit := #Auxiliares.A3)
      I_Contact( #Auxiliares.A2 )
      wire#w1
      Coil( #Instancia_Valvula.alarma )
   END_RUNG
   RUNG wire#w1
      Coil( #AlarmaStruct )
   END_RUNG
   // the same network as SCL:
   #_w1 := NOT #TemporizadorAlarma.Q AND #Auxiliares.A3;   // falling edge of #TemporizadorAlarma.Q
   #Auxiliares.A3 := #TemporizadorAlarma.Q;
   #Instancia_Valvula.alarma := #_w1 AND NOT #Auxiliares.A2;
   #AlarmaStruct := #Instancia_Valvula.alarma;
END_REGION
END_FUNCTION_BLOCK

FUNCTION_BLOCK "AlarmasDosificadoras"   // FB6, LAD
{ S7_Optimized_Access := 'TRUE' }
VERSION : 0.1
   VAR_OUTPUT
      AlarmaStruct : Bool;
   END_VAR
   VAR_IN_OUT
      Instancia_Valvula : "UDT_BOMBAS_DOSIFICADORAS";
   END_VAR
   VAR
      TemporizadorAlarma : TP_TIME;
      Auxiliares : Struct
         A1 : Bool;
         A2 : Bool;
         A3 : Bool;
         A4 : Bool;
         A5 : Bool;
         A6 : Bool;
         A7 : Bool;
      END_STRUCT;
   END_VAR
   VAR_TEMP   // added for the SCL form of the ladder/FBD networks
      _w1 : Bool;
      _w2 : Bool;
      _w3 : Bool;
      _w4 : Bool;
      _w5 : Bool;
   END_VAR
BEGIN

REGION Network 1
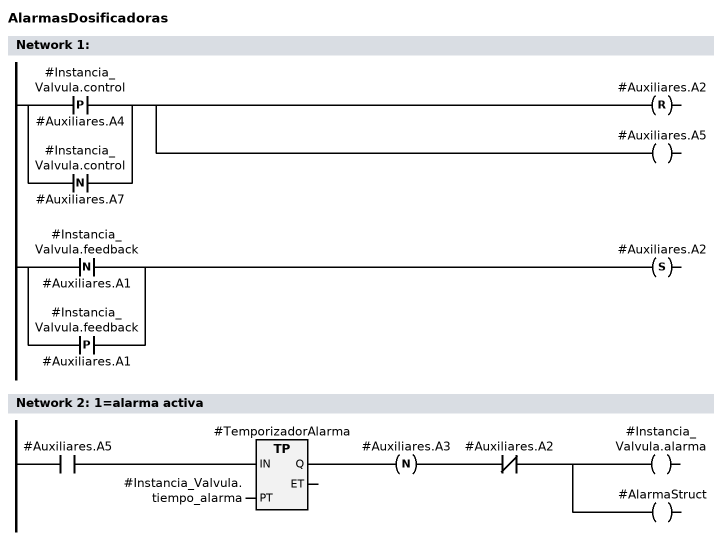
   RUNG wire#powerrail
      P_Contact(operand := #Instancia_Valvula.control, bit := #Auxiliares.A4)
      wire#w1
      R_Coil( #Auxiliares.A2 )
   END_RUNG
   RUNG wire#powerrail
      N_Contact(operand := #Instancia_Valvula.control, bit := #Auxiliares.A7)
   END_RUNG wire#w1
   RUNG wire#w1
      Coil( #Auxiliares.A5 )
   END_RUNG
   RUNG wire#powerrail
      N_Contact(operand := #Instancia_Valvula.feedback, bit := #Auxiliares.A1)
      wire#w2
      S_Coil( #Auxiliares.A2 )
   END_RUNG
   RUNG wire#powerrail
      P_Contact(operand := #Instancia_Valvula.feedback, bit := #Auxiliares.A1)
   END_RUNG wire#w2
   // the same network as SCL:
   #_w1 := #Instancia_Valvula.control AND NOT #Auxiliares.A4;   // rising edge of #Instancia_Valvula.control
   #Auxiliares.A4 := #Instancia_Valvula.control;
   #_w2 := NOT #Instancia_Valvula.control AND #Auxiliares.A7;   // falling edge of #Instancia_Valvula.control
   #Auxiliares.A7 := #Instancia_Valvula.control;
   #_w3 := #_w1 OR #_w2;
   IF #_w3 THEN #Auxiliares.A2 := FALSE; END_IF;
   #Auxiliares.A5 := #_w3;
   #_w4 := NOT #Instancia_Valvula.feedback AND #Auxiliares.A1;   // falling edge of #Instancia_Valvula.feedback
   #Auxiliares.A1 := #Instancia_Valvula.feedback;
   #_w5 := #Instancia_Valvula.feedback AND NOT #Auxiliares.A1;   // rising edge of #Instancia_Valvula.feedback
   #Auxiliares.A1 := #Instancia_Valvula.feedback;
   IF #_w4 OR #_w5 THEN #Auxiliares.A2 := TRUE; END_IF;
END_REGION

REGION Network 2: 1=alarma activa
   #TemporizadorAlarma(IN := #Auxiliares.A5, PT := #Instancia_Valvula.tiempo_alarma);   // TP
   #_w1 := NOT #TemporizadorAlarma.Q AND #Auxiliares.A3;   // falling edge
   #Auxiliares.A3 := #TemporizadorAlarma.Q;
   #Instancia_Valvula.alarma := #_w1 AND NOT #Auxiliares.A2;
   #AlarmaStruct := #Instancia_Valvula.alarma;
END_REGION
END_FUNCTION_BLOCK

FUNCTION_BLOCK "AlarmaPresionDiferencial"   // FB10, LAD
{ S7_Optimized_Access := 'TRUE' }
VERSION : 0.1
   VAR_OUTPUT
      PresionALcanzada : Bool;
   END_VAR
   VAR_IN_OUT
      SensorPT10 : "UDT_SENSORES_PRESION";
      SensorPT11 : "UDT_SENSORES_PRESION";
      Diferencial : "UDT_PRESION_DIFERENCIAL";
   END_VAR
   VAR
      Resultado : Int;
   END_VAR
BEGIN

REGION Network 1
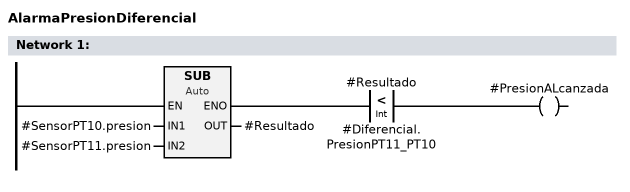
   RUNG wire#powerrail
      Sub(in1 := #SensorPT10.presion, in2 := #SensorPT11.presion, out => #Resultado)
      { S7_Templates := "SrcType := Int" } LT_Contact(in1 := #Resultado, in2 := #Diferencial.PresionPT11_PT10)
      Coil( #PresionALcanzada )
   END_RUNG
   // the same network as SCL:
   #Resultado := #SensorPT10.presion - #SensorPT11.presion;
   #PresionALcanzada := #Resultado < #Diferencial.PresionPT11_PT10;
END_REGION
END_FUNCTION_BLOCK

FUNCTION_BLOCK "AlarmasSensoresEspeciales"   // FB11, LAD
{ S7_Optimized_Access := 'TRUE' }
VERSION : 0.1
   VAR_OUTPUT
      AlarmaStruct_Alto : Bool;
      AlarmaStruct_Bajo : Bool;
      FallaGeneral : Bool;
   END_VAR
   VAR_IN_OUT
      Sensor : "UDT_SENSORES_ESPECIALES";
   END_VAR
BEGIN

REGION Network 1
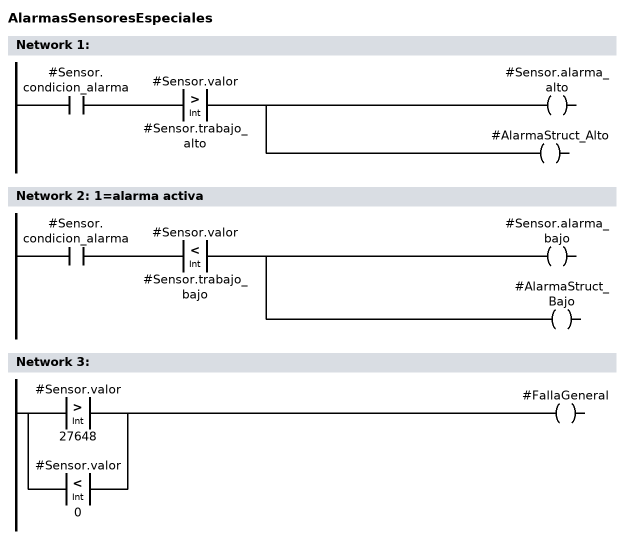
   RUNG wire#powerrail
      Contact( #Sensor.condicion_alarma )
      { S7_Templates := "SrcType := Int" } GT_Contact(in1 := #Sensor.valor, in2 := #Sensor.trabajo_alto)
      wire#w1
      Coil( #Sensor.alarma_alto )
   END_RUNG
   RUNG wire#w1
      Coil( #AlarmaStruct_Alto )
   END_RUNG
   // the same network as SCL:
   #Sensor.alarma_alto := #Sensor.condicion_alarma AND (#Sensor.valor > #Sensor.trabajo_alto);
   #AlarmaStruct_Alto := #Sensor.alarma_alto;
END_REGION

REGION Network 2: 1=alarma activa
   RUNG wire#powerrail
      Contact( #Sensor.condicion_alarma )
      { S7_Templates := "SrcType := Int" } LT_Contact(in1 := #Sensor.valor, in2 := #Sensor.trabajo_bajo)
      wire#w1
      Coil( #Sensor.alarma_bajo )
   END_RUNG
   RUNG wire#w1
      Coil( #AlarmaStruct_Bajo )
   END_RUNG
   // the same network as SCL:
   #Sensor.alarma_bajo := #Sensor.condicion_alarma AND (#Sensor.valor < #Sensor.trabajo_bajo);
   #AlarmaStruct_Bajo := #Sensor.alarma_bajo;
END_REGION

REGION Network 3
   RUNG wire#powerrail
      { S7_Templates := "SrcType := Int" } GT_Contact(in1 := #Sensor.valor, in2 := 27648)
      wire#w1
      Coil( #FallaGeneral )
   END_RUNG
   RUNG wire#powerrail
      { S7_Templates := "SrcType := Int" } LT_Contact(in1 := #Sensor.valor, in2 := 0)
   END_RUNG wire#w1
   // the same network as SCL:
   #FallaGeneral := (#Sensor.valor > 27648) OR (#Sensor.valor < 0);
END_REGION
END_FUNCTION_BLOCK

FUNCTION_BLOCK "AlarmasFlujo"   // FB12, LAD
{ S7_Optimized_Access := 'TRUE' }
VERSION : 0.1
   VAR_OUTPUT
      AlarmaStruct_Alto : Bool;
      AlarmaStruct_Bajo : Bool;
      FallaGeneral : Bool;
   END_VAR
   VAR_IN_OUT
      Sensor : "UDT_SENSORES_FLUJO";
   END_VAR
BEGIN

REGION Network 1
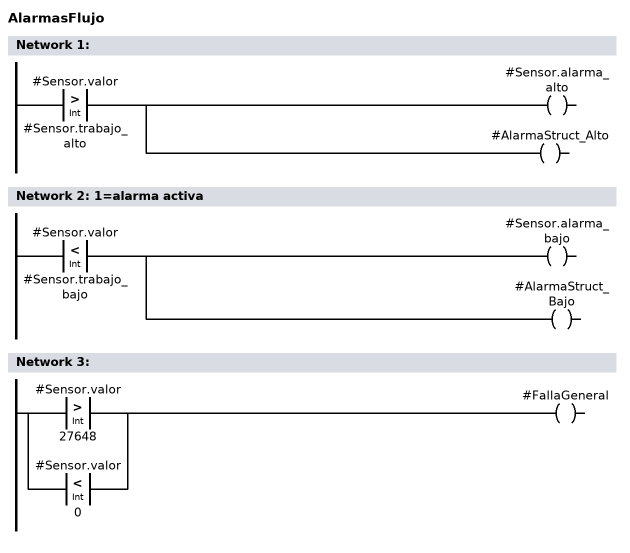
   RUNG wire#powerrail
      { S7_Templates := "SrcType := Int" } GT_Contact(in1 := #Sensor.valor, in2 := #Sensor.trabajo_alto)
      wire#w1
      Coil( #Sensor.alarma_alto )
   END_RUNG
   RUNG wire#w1
      Coil( #AlarmaStruct_Alto )
   END_RUNG
   // the same network as SCL:
   #Sensor.alarma_alto := #Sensor.valor > #Sensor.trabajo_alto;
   #AlarmaStruct_Alto := #Sensor.alarma_alto;
END_REGION

REGION Network 2: 1=alarma activa
   RUNG wire#powerrail
      { S7_Templates := "SrcType := Int" } LT_Contact(in1 := #Sensor.valor, in2 := #Sensor.trabajo_bajo)
      wire#w1
      Coil( #Sensor.alarma_bajo )
   END_RUNG
   RUNG wire#w1
      Coil( #AlarmaStruct_Bajo )
   END_RUNG
   // the same network as SCL:
   #Sensor.alarma_bajo := #Sensor.valor < #Sensor.trabajo_bajo;
   #AlarmaStruct_Bajo := #Sensor.alarma_bajo;
END_REGION

REGION Network 3
   RUNG wire#powerrail
      { S7_Templates := "SrcType := Int" } GT_Contact(in1 := #Sensor.valor, in2 := 27648)
      wire#w1
      Coil( #FallaGeneral )
   END_RUNG
   RUNG wire#powerrail
      { S7_Templates := "SrcType := Int" } LT_Contact(in1 := #Sensor.valor, in2 := 0)
   END_RUNG wire#w1
   // the same network as SCL:
   #FallaGeneral := (#Sensor.valor > 27648) OR (#Sensor.valor < 0);
END_REGION
END_FUNCTION_BLOCK

FUNCTION_BLOCK "AlarmasPresioOsmosis"   // FB13, LAD
{ S7_Optimized_Access := 'TRUE' }
VERSION : 0.1
   VAR_OUTPUT
      AlarmaStruct_Alto : Bool;
      AlarmaStruct_Bajo : Bool;
   END_VAR
   VAR_IN_OUT
      SensorPresion : "UDT_SENSORES_PRESION";
   END_VAR
BEGIN

REGION Network 1
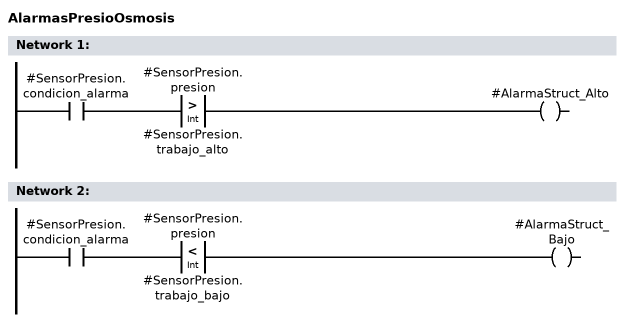
   RUNG wire#powerrail
      Contact( #SensorPresion.condicion_alarma )
      { S7_Templates := "SrcType := Int" } GT_Contact(in1 := #SensorPresion.presion, in2 := #SensorPresion.trabajo_alto)
      Coil( #AlarmaStruct_Alto )
   END_RUNG
   // the same network as SCL:
   #AlarmaStruct_Alto := #SensorPresion.condicion_alarma AND (#SensorPresion.presion > #SensorPresion.trabajo_alto);
END_REGION

REGION Network 2
   RUNG wire#powerrail
      Contact( #SensorPresion.condicion_alarma )
      { S7_Templates := "SrcType := Int" } LT_Contact(in1 := #SensorPresion.presion, in2 := #SensorPresion.trabajo_bajo)
      Coil( #AlarmaStruct_Bajo )
   END_RUNG
   // the same network as SCL:
   #AlarmaStruct_Bajo := #SensorPresion.condicion_alarma AND (#SensorPresion.presion < #SensorPresion.trabajo_bajo);
END_REGION
END_FUNCTION_BLOCK

FUNCTION_BLOCK "AlarmasFlujoDiferencial"   // FB14, LAD
{ S7_Optimized_Access := 'TRUE' }
VERSION : 0.1
   VAR_IN_OUT
      SensorFI08FI10 : "UDT_SENSORES_NIVEL";
   END_VAR
   VAR
      Resultado : Bool;
      PresionAlcanzada : Bool;
   END_VAR
BEGIN
END_FUNCTION_BLOCK

ORGANIZATION_BLOCK "Main_Alarmas"   // OB124, LAD, ProgramCycle
TITLE = "Main Program Sweep (Cycle)"
{ S7_Optimized_Access := 'TRUE' }
VERSION : 0.1
   VAR_INPUT
      Initial_Call : Bool;   // Initial call of this OB
      Remanence : Bool;   // =True, if remanent data are available
   END_VAR
BEGIN

REGION Network 1
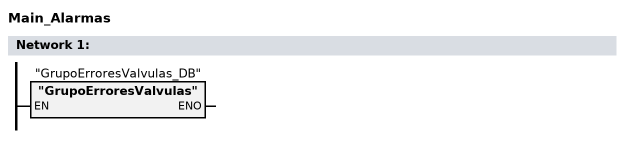
   RUNG wire#powerrail
      "GrupoErroresValvulas_DB"()
   END_RUNG
   // the same network as SCL:
   "GrupoErroresValvulas_DB"();   // "GrupoErroresValvulas"
END_REGION
END_ORGANIZATION_BLOCK

// folder: Asignaciones

FUNCTION_BLOCK "Horometria"   // FB9, LAD
{ S7_Optimized_Access := 'TRUE' }
VERSION : 0.1
BEGIN
END_FUNCTION_BLOCK

FUNCTION_BLOCK "PresionANivel"   // FB16, LAD
{ S7_Optimized_Access := 'TRUE' }
VERSION : 0.1
BEGIN
END_FUNCTION_BLOCK

FUNCTION "Asignaciones_Totales" : Void   // FC1, SCL
{ S7_Optimized_Access := 'TRUE' }
VERSION : 0.1
BEGIN
   //Entradas
   "UDT_Objetos".Auxiliares.AuxiliaresGenerales.Vigilante_Tension := "KF1_feedback";
   "UDT_Objetos".Auxiliares.AuxiliaresGenerales.Paro_Emergencia := "S1_feedback";
   "UDT_Objetos".Bombas."BC-08".feedback := "BC-08_feedback";
   "UDT_Objetos".Bombas."BC-09".feedback := "BC-09_feedback";
   "UDT_Objetos".Bombas."BC-10".feedback := "BC-10_feedback";
   "UDT_Objetos".Bombas."BC-11".feedback := "BC-11_feedback_protector";
   "UDT_Objetos".Bombas."BC-11".alarma_variador := "BC-11_feedback_variador";
   "UDT_Objetos".Bombas."BC-12".feedback := "BC-12_feedback";
   "UDT_Objetos".Bombas."BC-13".feedback := "BC-13_feedback";
   "UDT_Objetos".Bombas."BC-14".feedback := "BC-14_feedback";
   "UDT_Objetos".Equipos_Especiales."BLW-01".feedback := "BLW-01_feedback";
   "UDT_Objetos".Equipos_Especiales."UV-01".feedback := "UV-01_feedback";
   "UDT_Objetos".Dosificadoras."BD-AI-01".feedback := "BD-AI-01_feedback";
   "UDT_Objetos".Dosificadoras."BD-BIO-01".feedback := "BD-BIO-01_feedback";
   "UDT_Objetos".Dosificadoras."BD-HIP-01".feedback := "BD-HIP-01_feedback";
   "UDT_Objetos".Dosificadoras."BD-HIP-02".feedback := "BD-HIP-02_feedback";
   "UDT_Objetos".Dosificadoras."BD-MBI-01".feedback := "BD-MBI-01_feedback";
   "UDT_Objetos".Dosificadoras."BD-UF-01".feedback := "BD-UF-01_feedback";
   "UDT_Objetos".Valvulas."VM-27".feedback := "VM-27-2_feedback";
   "UDT_Objetos".Valvulas."VM-29".feedback := "VM-29_feedback";
   "UDT_Objetos".Valvulas."VM-31".feedback := "VM-31_feedback";
   "UDT_Objetos".Valvulas."VM-32".feedback := "VM-32_feedback";
   "UDT_Objetos".Valvulas."VM-33".feedback := "VM-33_feedback";
   "UDT_Objetos".Valvulas."VM-34".feedback := "VM-34_feedback";
   "UDT_Objetos".Valvulas."VM-35".feedback := "VM-35_feedback";
   "UDT_Objetos".Valvulas."VM-36".feedback := "VM-36_feedback";
   "UDT_Objetos".Valvulas."VM-39".feedback := "VM-39_feedback";
   "UDT_Objetos".Valvulas."VM-40".feedback := "VM-40_feedback";
   "UDT_Objetos".Valvulas."VM-41".feedback := "VM-41_feedback";
   "UDT_Objetos".Valvulas."VM-42".feedback := "VM-42_feedback";
   "UDT_Objetos".Valvulas."VM-45".feedback := "VM-45_feedback";
   "UDT_Objetos".Valvulas."VM-46".feedback := "VM-46_feedback";
   "UDT_Objetos".Valvulas."VM-47".feedback := "VM-47_feedback";
   "UDT_Objetos".Valvulas."VM-48".feedback := "VM-48_feedback";
   "UDT_Objetos".Valvulas."VM-49".feedback := "VM-49_feedback";
   "UDT_Objetos".Valvulas."VM-50".feedback := "VM-50_feedback";
   "UDT_Objetos".Valvulas."VM-51".feedback := "VM-51_feedback";
   "UDT_Objetos".Valvulas."VM-52".feedback := "VM-52_feedback";
   "UDT_Objetos".Valvulas."VM-53".feedback := "VM-53_feedback";
   "UDT_Objetos".Valvulas."VM-56".feedback := "VM-56_feedback";
   "UDT_Objetos".Valvulas."VM-57".feedback := "VM-57_feedback";
   "UDT_Objetos".Valvulas."VM-58".feedback := "VM-58_feedback";
   "UDT_Objetos".Valvulas."VM-61".feedback := "VM-61_feedback";
   "UDT_Objetos".Valvulas."VM-62".feedback := "VM-62_feedback";
   "UDT_Objetos".Valvulas."VM-63".feedback := "VM-63_feedback";
   "UDT_Objetos".Dosificadoras."BD-HIP-01".nivel_bajo_quimico := "LSL-03_feedback";
   "UDT_Objetos".Dosificadoras."BD-MBI-01".nivel_bajo_quimico :="LSL-04_feedback";
   "UDT_Objetos".Dosificadoras."BD-AI-01".nivel_bajo_quimico :="LSL-05_feedback";
   "UDT_Objetos".Dosificadoras."BD-BIO-01".nivel_bajo_quimico :="LSL-07_feedback";
   "UDT_Objetos".Dosificadoras."BD-HIP-02".nivel_bajo_quimico :="LSL-08_feedback";
   "UDT_Objetos".Dosificadoras."BD-UF-01".nivel_bajo_quimico :="LSL-XX_feedback";
   "UDT_Objetos".Sensores_Especiales."COT-01".valor := "COT-01_feedback";
   "UDT_Objetos".Sensores_Especiales."CT-02".valor := "CT-02_feedback";
   "UDT_Objetos".Sensores_Especiales."ORP-01".valor := "ORP-01_feedback";
   "UDT_Objetos".Sensores_Especiales."ORP-02".valor := "ORP-02_feedback";
   "UDT_Objetos".Sensores_Especiales."PH-04".valor := "PH-04_feedback";
   "UDT_Objetos".Sensores_Especiales."TRB-02".valor := "TRB-02_feedback";
   "UDT_Objetos".Flujo."FI-06".valor := "FI-06_feedback";
   "UDT_Objetos".Flujo."FI-07".valor := "FI-07_feedback";
   "UDT_Objetos".Flujo."FI-08".valor := "FI-08_feedback";
   "UDT_Objetos".Flujo."FI-09".valor := "FI-09_feedback";
   "UDT_Objetos".Flujo."FI-10".valor := "FI-10_feedback";
   "UDT_Objetos".Flujo."FI-11".valor := "FI-11_feedback";
   "UDT_Objetos".Presion."PT-05".valor := "PT-05_feedback";
   "UDT_Objetos".Presion."PT-06".valor := "PT-06_feedback";
   "UDT_Objetos".Nivel."PT-07".valor := "PT-07_feedback";
   "UDT_Objetos".Presion."PT-08".valor := "PT-08_feedback";
   "UDT_Objetos".Presion."PT-09".valor := "PT-09_feedback";
   "UDT_Objetos".Presion."PT-10".valor := "PT-10_feedback";
   "UDT_Objetos".Presion."PT-11".valor := "PT-11_feedback";
   "UDT_Objetos".Nivel."PT-12".valor := "PT-12_feedback";
   "UDT_Objetos".Nivel."PT-13".valor := "PT-13_feedback";
   "UDT_Objetos".Nivel."LSH-02".alarma_nivel:= "LSH-02_feedback";
   "UDT_Objetos".Nivel."LSH-EX1".alarma_nivel := "LSH-EX1_feedback";
   "UDT_Objetos".Nivel."LSL-06".alarma_nivel := "LSL-06_feedback";
   "UDT_Objetos".Nivel."RAD-04".valor := "RAD-04_feedback";
   "UDT_Objetos".Nivel."RAD-05".valor := "RAD-05_feedback";
   "UDT_Objetos".Nivel."RAD-06".valor := "RAD-06_feedback";

   //Salidas
   "BC-08_control" := "UDT_Objetos".Bombas."BC-08".control;
   "BC-09_control" := "UDT_Objetos".Bombas."BC-09".control;
   "BC-10_control" := "UDT_Objetos".Bombas."BC-10".control;
   "BC-11_control" := "UDT_Objetos".Bombas."BC-11".control;
   "BC-11_frecuencia" := "UDT_Objetos".Bombas."BC-11".valor;
   "BC-12_control" := "UDT_Objetos".Bombas."BC-12".control;
   "BC-13_control" := "UDT_Objetos".Bombas."BC-13".control;
   "BC-14_control" := "UDT_Objetos".Bombas."BC-14".control;
   "BLW-01_control" := "UDT_Objetos".Equipos_Especiales."BLW-01".control;
   "UV-01_control" := "UDT_Objetos".Equipos_Especiales."UV-01".control;
   "BD-AI-01_control" := "UDT_Objetos".Dosificadoras."BD-AI-01".control;
   "BD-BIO-01_control" := "UDT_Objetos".Dosificadoras."BD-BIO-01".control;
   "BD-HIP-01_control" := "UDT_Objetos".Dosificadoras."BD-HIP-01".control;
   "BD-HIP-02_control" := "UDT_Objetos".Dosificadoras."BD-HIP-02".control;
   "BD-MBI-01_control" := "UDT_Objetos".Dosificadoras."BD-MBI-01".control;
   "BD-UF-01_control" := "UDT_Objetos".Dosificadoras."BD-UF-01".control;
   "VM-27-2_control" := "UDT_Objetos".Valvulas."VM-27".control;
   "VM-29_control" := "UDT_Objetos".Valvulas."VM-29".control;
   "VM-31_control" := "UDT_Objetos".Valvulas."VM-31".control;
   "VM-32_control" := "UDT_Objetos".Valvulas."VM-32".control;
   "VM-33_control" := "UDT_Objetos".Valvulas."VM-33".control;
   "VM-34_control" := "UDT_Objetos".Valvulas."VM-34".control;
   "VM-35_control" := "UDT_Objetos".Valvulas."VM-35".control;
   "VM-36_control" := "UDT_Objetos".Valvulas."VM-36".control;
   "VM-39_control" := "UDT_Objetos".Valvulas."VM-39".control;
   "VM-40_control" := "UDT_Objetos".Valvulas."VM-40".control;
   "VM-41_control" := "UDT_Objetos".Valvulas."VM-41".control;
   "VM-42_control" := "UDT_Objetos".Valvulas."VM-42".control;
   "VM-45_control" := "UDT_Objetos".Valvulas."VM-45".control;
   "VM-46_control" := "UDT_Objetos".Valvulas."VM-46".control;
   "VM-47_control" := "UDT_Objetos".Valvulas."VM-47".control;
   "VM-48_control" := "UDT_Objetos".Valvulas."VM-48".control;
   "VM-49_control" := "UDT_Objetos".Valvulas."VM-49".control;
   "VM-50_control" := "UDT_Objetos".Valvulas."VM-50".control;
   "VM-51_control" := "UDT_Objetos".Valvulas."VM-51".control;
   "VM-52_control" := "UDT_Objetos".Valvulas."VM-52".control;
   "VM-53_control" := "UDT_Objetos".Valvulas."VM-53".control;
   "VM-56_control" := "UDT_Objetos".Valvulas."VM-56".control;
   "VM-57_control" := "UDT_Objetos".Valvulas."VM-57".control;
   "VM-58_control" := "UDT_Objetos".Valvulas."VM-58".control;
   "VM-61_control" := "UDT_Objetos".Valvulas."VM-61".control;
   "VM-62_control" := "UDT_Objetos".Valvulas."VM-62".control;
   "VM-63_control" := "UDT_Objetos".Valvulas."VM-63".control;
END_FUNCTION

ORGANIZATION_BLOCK "Asignaciones"   // OB123, LAD, ProgramCycle
TITLE = "Main Program Sweep (Cycle)"
{ S7_Optimized_Access := 'TRUE' }
VERSION : 0.1
   VAR_INPUT
      Initial_Call : Bool;   // Initial call of this OB
      Remanence : Bool;   // =True, if remanent data are available
   END_VAR
BEGIN

REGION Network 1
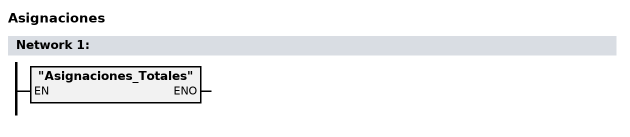
   RUNG wire#powerrail
      "Asignaciones_Totales"()
   END_RUNG
   // the same network as SCL:
   "Asignaciones_Totales"();
END_REGION
END_ORGANIZATION_BLOCK

// folder: Estados

FUNCTION_BLOCK "AsignacionesValvulas"   // FB3, LAD
{ S7_Optimized_Access := 'TRUE' }
VERSION : 0.1
   VAR_IN_OUT
      Valvula : "UDT_VALVULA_NEUMATICA";
   END_VAR
   VAR
      Auxiliares : Struct
         A1 : Bool;
         A2 : Bool;
         A3 : Bool;
         A4 : Bool;
         A5 : Bool;
      END_STRUCT;
   END_VAR
   VAR_TEMP   // added for the SCL form of the ladder/FBD networks
      _w1 : Bool;
      _w2 : Bool;
      _w3 : Bool;
   END_VAR
BEGIN

REGION Network 1
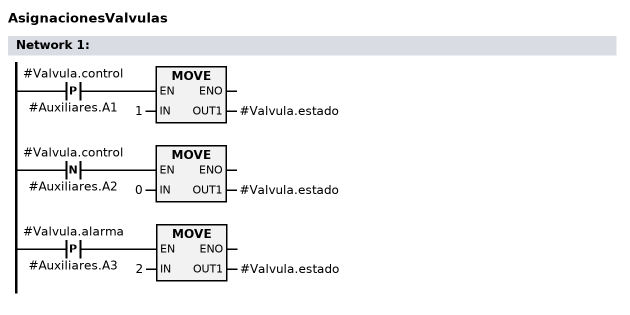
   RUNG wire#powerrail
      P_Contact(operand := #Valvula.control, bit := #Auxiliares.A1)
      Move(in := 1, out1 => #Valvula.estado)
   END_RUNG
   RUNG wire#powerrail
      N_Contact(operand := #Valvula.control, bit := #Auxiliares.A2)
      Move(in := 0, out1 => #Valvula.estado)
   END_RUNG
   RUNG wire#powerrail
      P_Contact(operand := #Valvula.alarma, bit := #Auxiliares.A3)
      Move(in := 2, out1 => #Valvula.estado)
   END_RUNG
   // the same network as SCL:
   #_w1 := #Valvula.control AND NOT #Auxiliares.A1;   // rising edge of #Valvula.control
   #Auxiliares.A1 := #Valvula.control;
   IF #_w1 THEN #Valvula.estado := 1; END_IF;
   #_w2 := NOT #Valvula.control AND #Auxiliares.A2;   // falling edge of #Valvula.control
   #Auxiliares.A2 := #Valvula.control;
   IF #_w2 THEN #Valvula.estado := 0; END_IF;
   #_w3 := #Valvula.alarma AND NOT #Auxiliares.A3;   // rising edge of #Valvula.alarma
   #Auxiliares.A3 := #Valvula.alarma;
   IF #_w3 THEN #Valvula.estado := 2; END_IF;
END_REGION
END_FUNCTION_BLOCK

FUNCTION_BLOCK "InstanciasValvulas"   // FB4, SCL
{ S7_Optimized_Access := 'TRUE' }
VERSION : 0.1
   VAR
      VM27 : "AsignacionesValvulas";
      VM29 : "AsignacionesValvulas";
      VM31 : "AsignacionesValvulas";
      VM32 : "AsignacionesValvulas";
      VM33 : "AsignacionesValvulas";
      VM34 : "AsignacionesValvulas";
      VM35 : "AsignacionesValvulas";
      VM36 : "AsignacionesValvulas";
      VM39 : "AsignacionesValvulas";
      VM40 : "AsignacionesValvulas";
      VM41 : "AsignacionesValvulas";
      VM42 : "AsignacionesValvulas";
      VM45 : "AsignacionesValvulas";
      VM46 : "AsignacionesValvulas";
      VM47 : "AsignacionesValvulas";
      VM48 : "AsignacionesValvulas";
      VM49 : "AsignacionesValvulas";
      VM50 : "AsignacionesValvulas";
      VM51 : "AsignacionesValvulas";
      VM52 : "AsignacionesValvulas";
      VM53 : "AsignacionesValvulas";
      VM56 : "AsignacionesValvulas";
      VM57 : "AsignacionesValvulas";
      VM58 : "AsignacionesValvulas";
      VM61 : "AsignacionesValvulas";
      VM62 : "AsignacionesValvulas";
      VM63 : "AsignacionesValvulas";
      BC08 : "AsignacionesBombas";
      BC09 : "AsignacionesBombas";
      BC10 : "AsignacionesBombas";
      BC11 : "AsignacionesBombas";
      BC12 : "AsignacionesBombas";
      BC13 : "AsignacionesBombas";
      BC14 : "AsignacionesBombas";
      BDI01 : "AsignacionesDosificadoras";
      BDIO01 : "AsignacionesDosificadoras";
      BDIP01 : "AsignacionesDosificadoras";
      BDIP02 : "AsignacionesDosificadoras";
      BDBI01 : "AsignacionesDosificadoras";
      BDF01 : "AsignacionesDosificadoras";
   END_VAR
BEGIN
   #VM27("UDT_Objetos".Valvulas."VM-27");
   #VM29("UDT_Objetos".Valvulas."VM-29");
   #VM31("UDT_Objetos".Valvulas."VM-31");
   #VM32("UDT_Objetos".Valvulas."VM-32");
   #VM33("UDT_Objetos".Valvulas."VM-33");
   #VM34("UDT_Objetos".Valvulas."VM-34");
   #VM35("UDT_Objetos".Valvulas."VM-35");
   #VM36("UDT_Objetos".Valvulas."VM-36");
   #VM39("UDT_Objetos".Valvulas."VM-39");
   #VM40("UDT_Objetos".Valvulas."VM-40");
   #VM41("UDT_Objetos".Valvulas."VM-41");
   #VM42("UDT_Objetos".Valvulas."VM-42");
   #VM45("UDT_Objetos".Valvulas."VM-45");
   #VM46("UDT_Objetos".Valvulas."VM-46");
   #VM47("UDT_Objetos".Valvulas."VM-47");
   #VM48("UDT_Objetos".Valvulas."VM-48");
   #VM49("UDT_Objetos".Valvulas."VM-49");
   #VM50("UDT_Objetos".Valvulas."VM-50");
   #VM51("UDT_Objetos".Valvulas."VM-51");
   #VM52("UDT_Objetos".Valvulas."VM-52");
   #VM53("UDT_Objetos".Valvulas."VM-53");
   #VM56("UDT_Objetos".Valvulas."VM-56");
   #VM57("UDT_Objetos".Valvulas."VM-57");
   #VM58("UDT_Objetos".Valvulas."VM-58");
   #VM61("UDT_Objetos".Valvulas."VM-61");
   #VM62("UDT_Objetos".Valvulas."VM-62");
   #VM63("UDT_Objetos".Valvulas."VM-63");
   #BC08("UDT_Objetos".Bombas."BC-08");
   #BC09("UDT_Objetos".Bombas."BC-09");
   #BC10("UDT_Objetos".Bombas."BC-10");
   #BC11("UDT_Objetos".Bombas."BC-11");
   #BC12("UDT_Objetos".Bombas."BC-12");
   #BC13("UDT_Objetos".Bombas."BC-13");
   #BC14("UDT_Objetos".Bombas."BC-14");
   #BDI01("UDT_Objetos".Dosificadoras."BD-AI-01");
   #BDIO01("UDT_Objetos".Dosificadoras."BD-BIO-01");
   #BDIP01("UDT_Objetos".Dosificadoras."BD-HIP-01");
   #BDIP02("UDT_Objetos".Dosificadoras."BD-HIP-02");
   #BDBI01("UDT_Objetos".Dosificadoras."BD-MBI-01");
   #BDF01("UDT_Objetos".Dosificadoras."BD-UF-01");
END_FUNCTION_BLOCK

FUNCTION_BLOCK "AsignacionesBombas"   // FB7, LAD
{ S7_Optimized_Access := 'TRUE' }
VERSION : 0.1
   VAR_IN_OUT
      Valvula : "UDT_BOMBAS";
   END_VAR
   VAR
      Auxiliares : Struct
         A1 : Bool;
         A2 : Bool;
         A3 : Bool;
         A4 : Bool;
         A5 : Bool;
      END_STRUCT;
   END_VAR
   VAR_TEMP   // added for the SCL form of the ladder/FBD networks
      _w1 : Bool;
      _w2 : Bool;
      _w3 : Bool;
   END_VAR
BEGIN

REGION Network 1
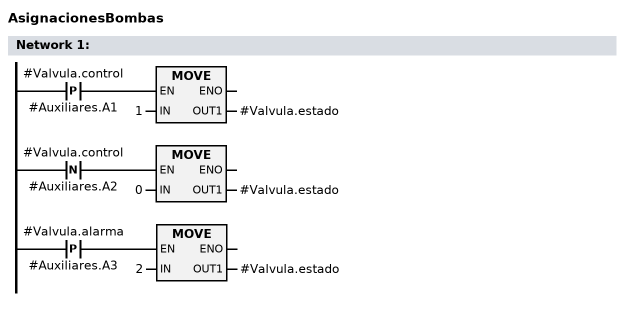
   RUNG wire#powerrail
      P_Contact(operand := #Valvula.control, bit := #Auxiliares.A1)
      Move(in := 1, out1 => #Valvula.estado)
   END_RUNG
   RUNG wire#powerrail
      N_Contact(operand := #Valvula.control, bit := #Auxiliares.A2)
      Move(in := 0, out1 => #Valvula.estado)
   END_RUNG
   RUNG wire#powerrail
      P_Contact(operand := #Valvula.alarma, bit := #Auxiliares.A3)
      Move(in := 2, out1 => #Valvula.estado)
   END_RUNG
   // the same network as SCL:
   #_w1 := #Valvula.control AND NOT #Auxiliares.A1;   // rising edge of #Valvula.control
   #Auxiliares.A1 := #Valvula.control;
   IF #_w1 THEN #Valvula.estado := 1; END_IF;
   #_w2 := NOT #Valvula.control AND #Auxiliares.A2;   // falling edge of #Valvula.control
   #Auxiliares.A2 := #Valvula.control;
   IF #_w2 THEN #Valvula.estado := 0; END_IF;
   #_w3 := #Valvula.alarma AND NOT #Auxiliares.A3;   // rising edge of #Valvula.alarma
   #Auxiliares.A3 := #Valvula.alarma;
   IF #_w3 THEN #Valvula.estado := 2; END_IF;
END_REGION
END_FUNCTION_BLOCK

FUNCTION_BLOCK "AsignacionesDosificadoras"   // FB8, LAD
{ S7_Optimized_Access := 'TRUE' }
VERSION : 0.1
   VAR_IN_OUT
      Valvula : "UDT_BOMBAS_DOSIFICADORAS";
   END_VAR
   VAR
      Auxiliares : Struct
         A1 : Bool;
         A2 : Bool;
         A3 : Bool;
         A4 : Bool;
         A5 : Bool;
      END_STRUCT;
   END_VAR
   VAR_TEMP   // added for the SCL form of the ladder/FBD networks
      _w1 : Bool;
      _w2 : Bool;
      _w3 : Bool;
   END_VAR
BEGIN

REGION Network 1
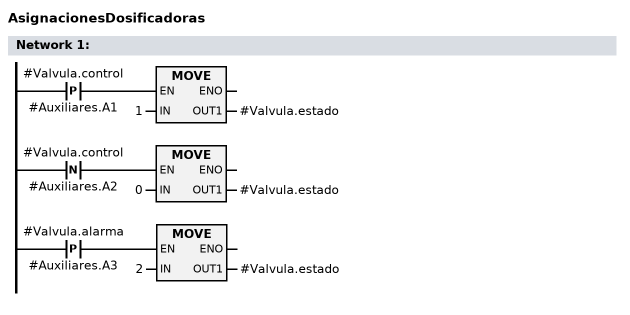
   RUNG wire#powerrail
      P_Contact(operand := #Valvula.control, bit := #Auxiliares.A1)
      Move(in := 1, out1 => #Valvula.estado)
   END_RUNG
   RUNG wire#powerrail
      N_Contact(operand := #Valvula.control, bit := #Auxiliares.A2)
      Move(in := 0, out1 => #Valvula.estado)
   END_RUNG
   RUNG wire#powerrail
      P_Contact(operand := #Valvula.alarma, bit := #Auxiliares.A3)
      Move(in := 2, out1 => #Valvula.estado)
   END_RUNG
   // the same network as SCL:
   #_w1 := #Valvula.control AND NOT #Auxiliares.A1;   // rising edge of #Valvula.control
   #Auxiliares.A1 := #Valvula.control;
   IF #_w1 THEN #Valvula.estado := 1; END_IF;
   #_w2 := NOT #Valvula.control AND #Auxiliares.A2;   // falling edge of #Valvula.control
   #Auxiliares.A2 := #Valvula.control;
   IF #_w2 THEN #Valvula.estado := 0; END_IF;
   #_w3 := #Valvula.alarma AND NOT #Auxiliares.A3;   // rising edge of #Valvula.alarma
   #Auxiliares.A3 := #Valvula.alarma;
   IF #_w3 THEN #Valvula.estado := 2; END_IF;
END_REGION
END_FUNCTION_BLOCK

ORGANIZATION_BLOCK "ManejoEstados"   // OB125, LAD, ProgramCycle
TITLE = "Main Program Sweep (Cycle)"
{ S7_Optimized_Access := 'TRUE' }
VERSION : 0.1
   VAR_INPUT
      Initial_Call : Bool;   // Initial call of this OB
      Remanence : Bool;   // =True, if remanent data are available
   END_VAR
BEGIN

REGION Network 1
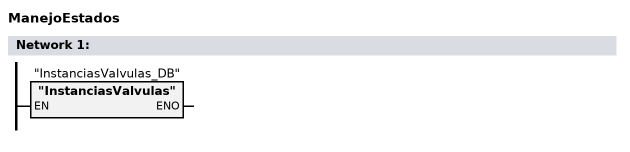
   RUNG wire#powerrail
      "InstanciasValvulas_DB"()
   END_RUNG
   // the same network as SCL:
   "InstanciasValvulas_DB"();   // "InstanciasValvulas"
END_REGION
END_ORGANIZATION_BLOCK

// folder: Procesos

FUNCTION_BLOCK "AutomaticoUF"   // FB15, LAD
{ S7_Optimized_Access := 'TRUE' }
VERSION : 0.1
   VAR
      MemoriasFlancos : Struct
         M0 : Bool;
         M1 : Bool;
         M2 : Bool;
      END_STRUCT;
      MemoriasGenerales : Struct
         M1 : Bool;
         M2 : Bool;
         M3 : Bool;
         M4 : Bool;
         M5 : Bool;
         M6 : Bool;
         M7 : Bool;
         M8 : Bool;
         M9 : Bool;
         "10" : Bool;
      END_STRUCT;
      T1 : "TiempoEspera";
      T2 : "TiempoEspera";
      T3 : "TiempoEspera";
      T4 : "TiempoEspera";
      T5 : "TiempoEspera";
      T6 : "TiempoEspera";
      T7 : "TiempoEspera";
      T8 : "TiempoEspera";
      T9 : "TiempoEspera";
      T10 : "TiempoEspera";
      TiempoPasoRetrolavado : TON_TIME;
      RetrolavadoActivo : Bool;
      R_TRIG_Instance : R_TRIG;
      IEC_Timer_0_Instance : TON_TIME;
      IEC_Timer_0_Instance_1 : TON_TIME;
      RetrolavadoActivo2 : Bool;
      TiempoEspera_Instance : "TiempoEspera";
      TiempoEspera_Instance_1 : "TiempoEspera";
      R_TRIG_Instance_1 : R_TRIG;
      F_TRIG_Instance : F_TRIG;
      R_TRIG_Instance_2 : R_TRIG;
      IEC_Timer_0_Instance_2 : TON_TIME;
      RetrolavadoActivo3 : Bool;
      IEC_Timer_0_Instance_3 : TON_TIME;
      RetrolavadoActivo4 : Bool;
      R_TRIG_Instance_3 : R_TRIG;
      R_TRIG_Instance_4 : R_TRIG;
      F_TRIG_Instance_1 : F_TRIG;
      TiempoEspera_Instance_2 : "TiempoEspera";
      R_TRIG_Instance_5 : R_TRIG;
      R_TRIG_Instance_6 : R_TRIG;
      R_TRIG_Instance_7 : R_TRIG;
      TiempoEspera_Instance_3 : "TiempoEspera";
      TiempoEspera_Instance_4 : "TiempoEspera";
      R_TRIG_Instance_8 : R_TRIG;
      R_TRIG_Instance_9 : R_TRIG;
      TiempoEspera_Instance_5 : "TiempoEspera";
      TiempoEspera_Instance_6 : "TiempoEspera";
      R_TRIG_Instance_10 : R_TRIG;
      TiempoEspera_Instance_7 : "TiempoEspera";
   END_VAR
   VAR_TEMP
      PT071 : Bool;
      PT072 : Bool;
      PT073 : Bool;
      PT074 : Bool;
   END_VAR
   VAR_TEMP   // added for the SCL form of the ladder/FBD networks
      _w1 : Bool;
      _w2 : Bool;
      _w3 : Bool;
      _w4 : Bool;
   END_VAR
BEGIN

REGION Network 1: RAD04 CONDICIONES
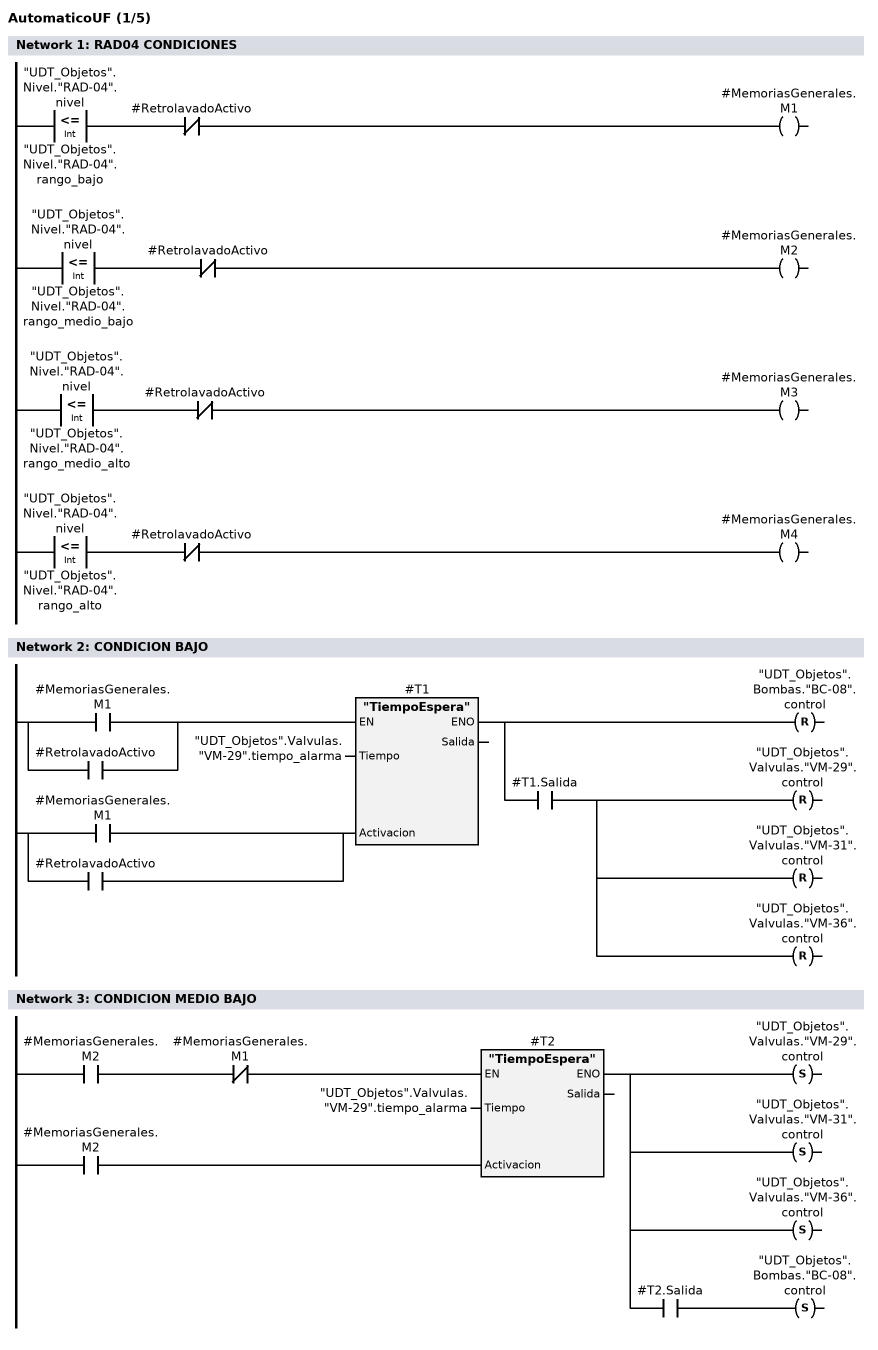
   RUNG wire#powerrail
      { S7_Templates := "SrcType := Int" } LE_Contact(in1 := "UDT_Objetos".Nivel."RAD-04".nivel, in2 := "UDT_Objetos".Nivel."RAD-04".rango_bajo)
      I_Contact( #RetrolavadoActivo )
      Coil( #MemoriasGenerales.M1 )
   END_RUNG
   RUNG wire#powerrail
      { S7_Templates := "SrcType := Int" } LE_Contact(in1 := "UDT_Objetos".Nivel."RAD-04".nivel, in2 := "UDT_Objetos".Nivel."RAD-04".rango_medio_bajo)
      I_Contact( #RetrolavadoActivo )
      Coil( #MemoriasGenerales.M2 )
   END_RUNG
   RUNG wire#powerrail
      { S7_Templates := "SrcType := Int" } LE_Contact(in1 := "UDT_Objetos".Nivel."RAD-04".nivel, in2 := "UDT_Objetos".Nivel."RAD-04".rango_medio_alto)
      I_Contact( #RetrolavadoActivo )
      Coil( #MemoriasGenerales.M3 )
   END_RUNG
   RUNG wire#powerrail
      { S7_Templates := "SrcType := Int" } LE_Contact(in1 := "UDT_Objetos".Nivel."RAD-04".nivel, in2 := "UDT_Objetos".Nivel."RAD-04".rango_alto)
      I_Contact( #RetrolavadoActivo )
      Coil( #MemoriasGenerales.M4 )
   END_RUNG
   // the same network as SCL:
   #MemoriasGenerales.M1 := ("UDT_Objetos".Nivel."RAD-04".nivel <= "UDT_Objetos".Nivel."RAD-04".rango_bajo) AND NOT #RetrolavadoActivo;
   #MemoriasGenerales.M2 := ("UDT_Objetos".Nivel."RAD-04".nivel <= "UDT_Objetos".Nivel."RAD-04".rango_medio_bajo) AND NOT #RetrolavadoActivo;
   #MemoriasGenerales.M3 := ("UDT_Objetos".Nivel."RAD-04".nivel <= "UDT_Objetos".Nivel."RAD-04".rango_medio_alto) AND NOT #RetrolavadoActivo;
   #MemoriasGenerales.M4 := ("UDT_Objetos".Nivel."RAD-04".nivel <= "UDT_Objetos".Nivel."RAD-04".rango_alto) AND NOT #RetrolavadoActivo;
END_REGION

REGION Network 2: CONDICION BAJO
   RUNG wire#powerrail
      Contact( #MemoriasGenerales.M1 )
      wire#w1
      #T1(Activacion := wire#w2, Tiempo := "UDT_Objetos".Valvulas."VM-29".tiempo_alarma, Salida =>)
      wire#w3
      R_Coil( "UDT_Objetos".Bombas."BC-08".control )
   END_RUNG
   RUNG wire#powerrail
      Contact( #RetrolavadoActivo )
   END_RUNG wire#w1
   RUNG wire#powerrail
      Contact( #MemoriasGenerales.M1 )
   END_RUNG wire#w2
   RUNG wire#powerrail
      Contact( #RetrolavadoActivo )
   END_RUNG wire#w2
   RUNG wire#w3
      Contact( #T1.Salida )
      wire#w4
      R_Coil( "UDT_Objetos".Valvulas."VM-29".control )
   END_RUNG
   RUNG wire#w4
      R_Coil( "UDT_Objetos".Valvulas."VM-31".control )
   END_RUNG
   RUNG wire#w4
      R_Coil( "UDT_Objetos".Valvulas."VM-36".control )
   END_RUNG
   // the same network as SCL:
   #T1(EN := #MemoriasGenerales.M1 OR #RetrolavadoActivo,   // "TiempoEspera"
       Tiempo := "UDT_Objetos".Valvulas."VM-29".tiempo_alarma,
       Activacion := #MemoriasGenerales.M1 OR #RetrolavadoActivo,
       ENO => #_w1);
   IF #_w1 THEN "UDT_Objetos".Bombas."BC-08".control := FALSE; END_IF;
   IF #_w1 AND #T1.Salida THEN
       "UDT_Objetos".Valvulas."VM-29".control := FALSE;
       "UDT_Objetos".Valvulas."VM-31".control := FALSE;
       "UDT_Objetos".Valvulas."VM-36".control := FALSE;
   END_IF;
END_REGION

REGION Network 3: CONDICION MEDIO BAJO
   RUNG wire#powerrail
      Contact( #MemoriasGenerales.M2 )
      I_Contact( #MemoriasGenerales.M1 )
      #T2(Activacion := wire#w1, Tiempo := "UDT_Objetos".Valvulas."VM-29".tiempo_alarma, Salida =>)
      wire#w2
      S_Coil( "UDT_Objetos".Valvulas."VM-29".control )
   END_RUNG
   RUNG wire#powerrail
      Contact( #MemoriasGenerales.M2 )
   END_RUNG wire#w1
   RUNG wire#w2
      S_Coil( "UDT_Objetos".Valvulas."VM-31".control )
   END_RUNG
   RUNG wire#w2
      S_Coil( "UDT_Objetos".Valvulas."VM-36".control )
   END_RUNG
   RUNG wire#w2
      Contact( #T2.Salida )
      S_Coil( "UDT_Objetos".Bombas."BC-08".control )
   END_RUNG
   // the same network as SCL:
   #T2(EN := #MemoriasGenerales.M2 AND NOT #MemoriasGenerales.M1,   // "TiempoEspera"
       Tiempo := "UDT_Objetos".Valvulas."VM-29".tiempo_alarma,
       Activacion := #MemoriasGenerales.M2,
       ENO => #_w1);
   IF #_w1 THEN
       "UDT_Objetos".Valvulas."VM-29".control := TRUE;
       "UDT_Objetos".Valvulas."VM-31".control := TRUE;
       "UDT_Objetos".Valvulas."VM-36".control := TRUE;
   END_IF;
   IF #_w1 AND #T2.Salida THEN "UDT_Objetos".Bombas."BC-08".control := TRUE; END_IF;
END_REGION

REGION Network 4: CONDICION MEDIO ALTO
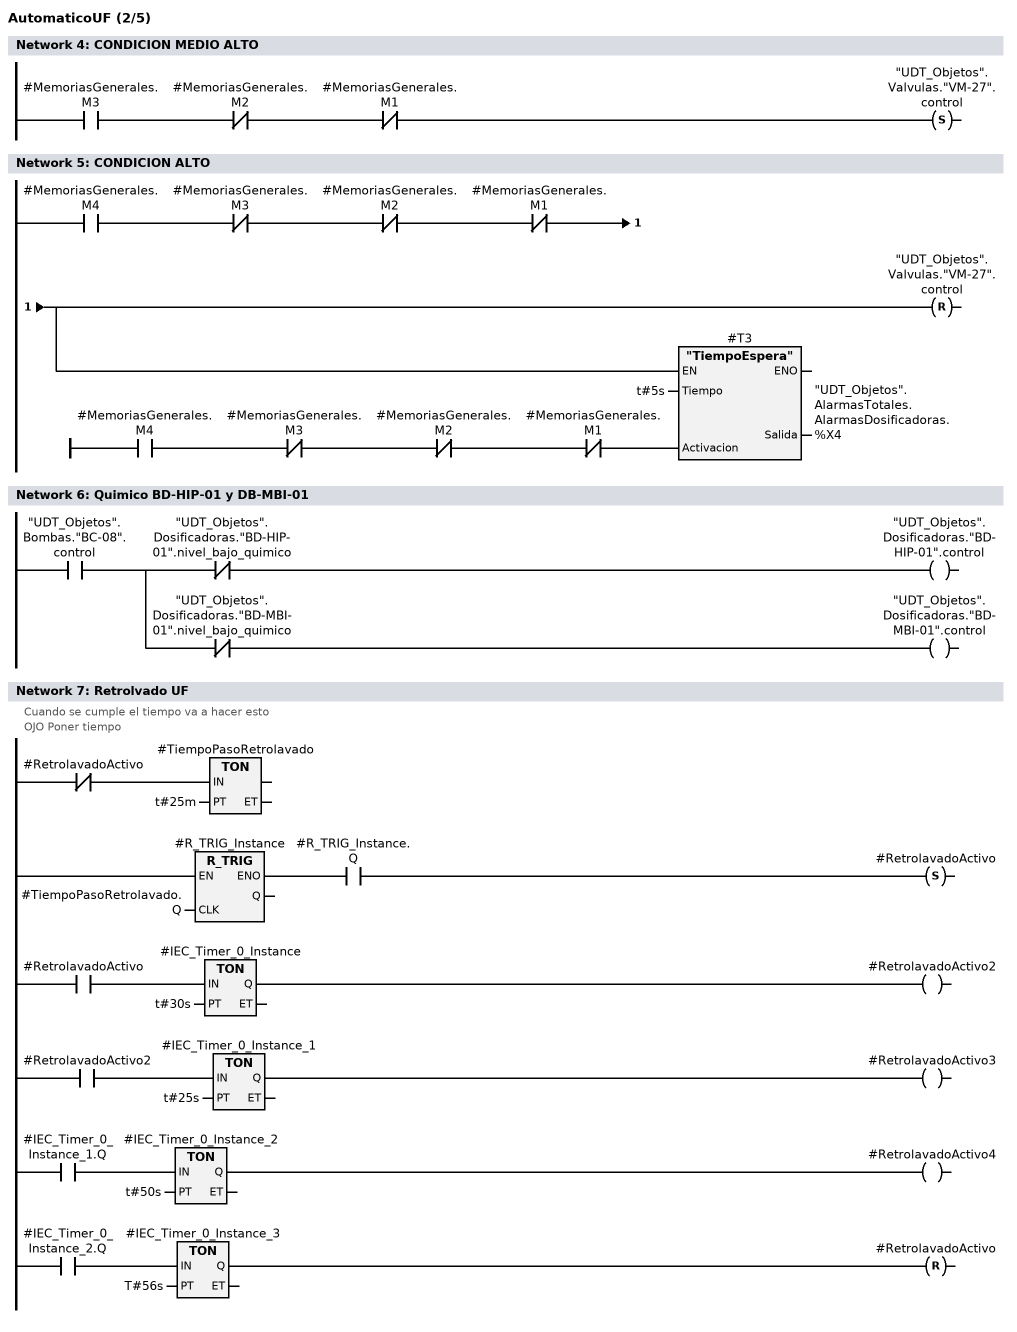
   RUNG wire#powerrail
      Contact( #MemoriasGenerales.M3 )
      I_Contact( #MemoriasGenerales.M2 )
      I_Contact( #MemoriasGenerales.M1 )
      S_Coil( "UDT_Objetos".Valvulas."VM-27".control )
   END_RUNG
   // the same network as SCL:
   IF #MemoriasGenerales.M3 AND NOT #MemoriasGenerales.M2 AND NOT #MemoriasGenerales.M1 THEN
       "UDT_Objetos".Valvulas."VM-27".control := TRUE;
   END_IF;
END_REGION

REGION Network 5: CONDICION ALTO
   RUNG wire#powerrail
      Contact( #MemoriasGenerales.M4 )
      I_Contact( #MemoriasGenerales.M3 )
      I_Contact( #MemoriasGenerales.M2 )
      I_Contact( #MemoriasGenerales.M1 )
      wire#w1
      R_Coil( "UDT_Objetos".Valvulas."VM-27".control )
   END_RUNG
   RUNG wire#w1
      #T3(Activacion := wire#w2, Tiempo := t#5s, Salida => "UDT_Objetos".AlarmasTotales.AlarmasDosificadoras.%X4)
   END_RUNG
   RUNG wire#powerrail
      Contact( #MemoriasGenerales.M4 )
      I_Contact( #MemoriasGenerales.M3 )
      I_Contact( #MemoriasGenerales.M2 )
      I_Contact( #MemoriasGenerales.M1 )
   END_RUNG wire#w2
   // the same network as SCL:
   IF #MemoriasGenerales.M4 AND NOT #MemoriasGenerales.M3 AND NOT #MemoriasGenerales.M2 AND NOT #MemoriasGenerales.M1 THEN
       "UDT_Objetos".Valvulas."VM-27".control := FALSE;
       #T3(Tiempo := t#5s,   // "TiempoEspera"
           Activacion := #MemoriasGenerales.M4 AND NOT #MemoriasGenerales.M3 AND NOT #MemoriasGenerales.M2 AND NOT #MemoriasGenerales.M1,
           Salida => "UDT_Objetos".AlarmasTotales.AlarmasDosificadoras.%X4);
   END_IF;
END_REGION

REGION Network 6: Quimico BD-HIP-01 y DB-MBI-01
   RUNG wire#powerrail
      Contact( "UDT_Objetos".Bombas."BC-08".control )
      wire#w1
      I_Contact( "UDT_Objetos".Dosificadoras."BD-HIP-01".nivel_bajo_quimico )
      Coil( "UDT_Objetos".Dosificadoras."BD-HIP-01".control )
   END_RUNG
   RUNG wire#w1
      I_Contact( "UDT_Objetos".Dosificadoras."BD-MBI-01".nivel_bajo_quimico )
      Coil( "UDT_Objetos".Dosificadoras."BD-MBI-01".control )
   END_RUNG
   // the same network as SCL:
   "UDT_Objetos".Dosificadoras."BD-HIP-01".control := "UDT_Objetos".Bombas."BC-08".control AND NOT "UDT_Objetos".Dosificadoras."BD-HIP-01".nivel_bajo_quimico;
   "UDT_Objetos".Dosificadoras."BD-MBI-01".control := "UDT_Objetos".Bombas."BC-08".control AND NOT "UDT_Objetos".Dosificadoras."BD-MBI-01".nivel_bajo_quimico;
END_REGION

REGION Network 7: Retrolvado UF
   // Cuando se cumple el tiempo va a hacer esto
   // OJO Poner tiempo
   // ENO of a box is taken as its EN; it also drops when the box reports an error
   #TiempoPasoRetrolavado(IN := NOT #RetrolavadoActivo, PT := t#25m);   // TON
   #R_TRIG_Instance(CLK := #TiempoPasoRetrolavado.Q);   // R_TRIG
   IF #R_TRIG_Instance.Q THEN #RetrolavadoActivo := TRUE; END_IF;
   #IEC_Timer_0_Instance(IN := #RetrolavadoActivo, PT := t#30s);   // TON
   #RetrolavadoActivo2 := #IEC_Timer_0_Instance.Q;
   #IEC_Timer_0_Instance_1(IN := #RetrolavadoActivo2, PT := t#25s);   // TON
   #RetrolavadoActivo3 := #IEC_Timer_0_Instance_1.Q;
   #IEC_Timer_0_Instance_2(IN := #IEC_Timer_0_Instance_1.Q, PT := t#50s);   // TON
   #RetrolavadoActivo4 := #IEC_Timer_0_Instance_2.Q;
   #IEC_Timer_0_Instance_3(IN := #IEC_Timer_0_Instance_2.Q, PT := T#56s);   // TON
   IF #IEC_Timer_0_Instance_3.Q THEN #RetrolavadoActivo := FALSE; END_IF;
END_REGION

REGION Network 8: encendido bc-09
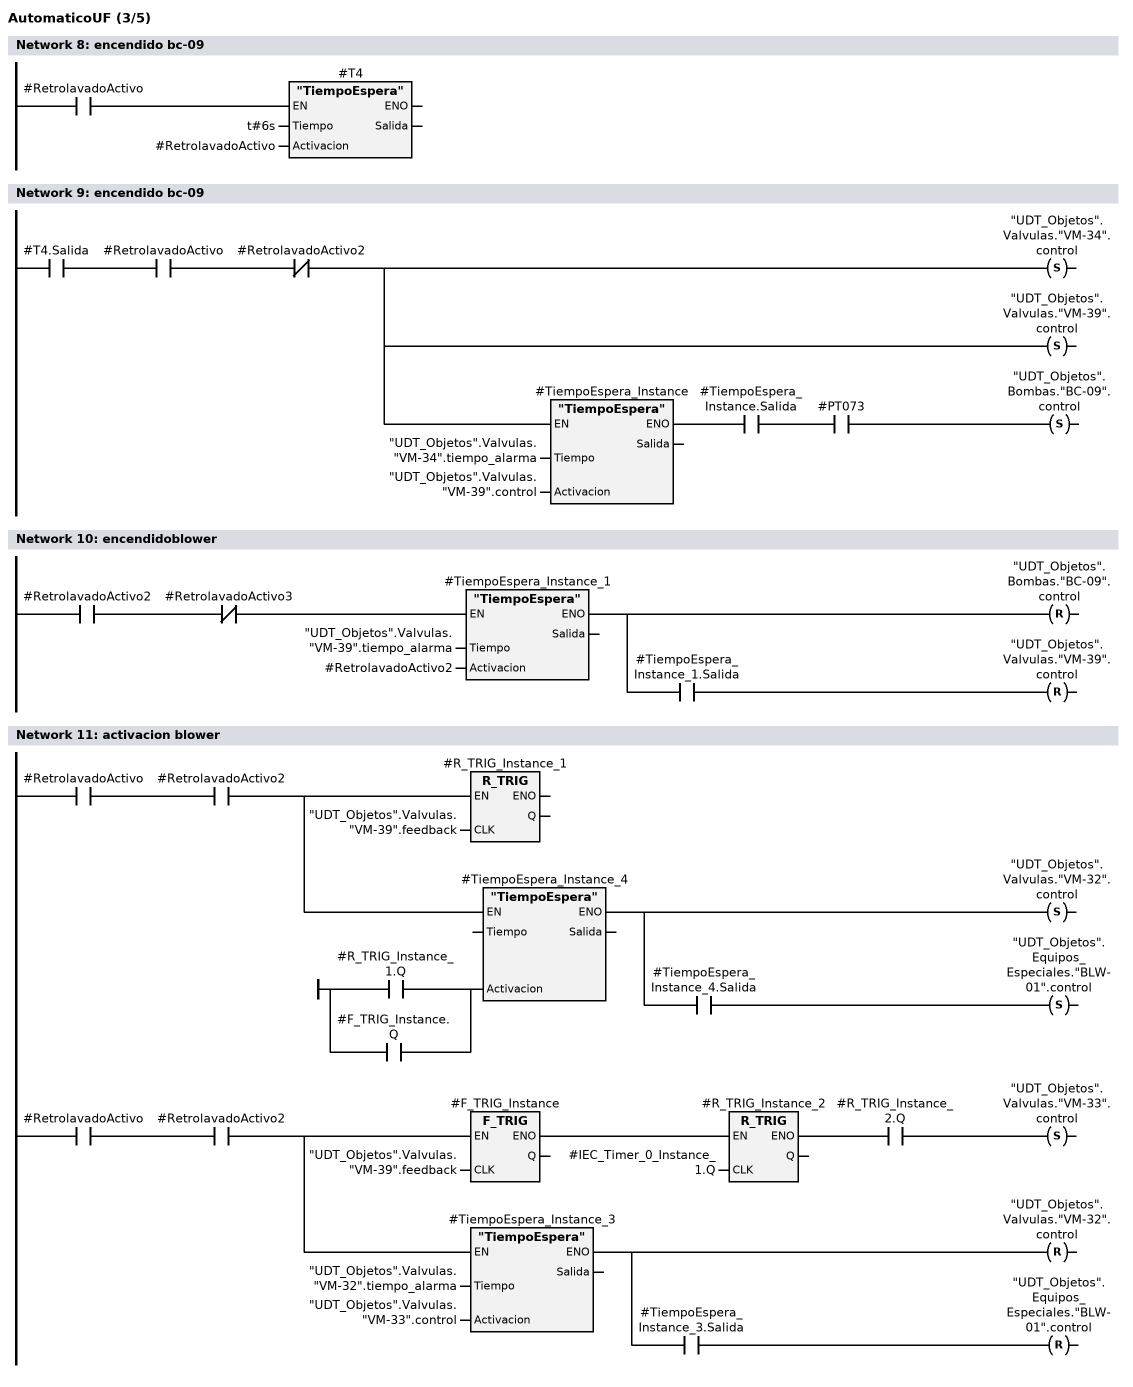
   RUNG wire#powerrail
      Contact( #RetrolavadoActivo )
      #T4(Tiempo := t#6s, Activacion := #RetrolavadoActivo, Salida =>)
   END_RUNG
   // the same network as SCL:
   IF #RetrolavadoActivo THEN
       #T4(Tiempo := t#6s, Activacion := #RetrolavadoActivo);   // "TiempoEspera"
   END_IF;
END_REGION

REGION Network 9: encendido bc-09
   RUNG wire#powerrail
      Contact( #T4.Salida )
      Contact( #RetrolavadoActivo )
      I_Contact( #RetrolavadoActivo2 )
      wire#w1
      S_Coil( "UDT_Objetos".Valvulas."VM-34".control )
   END_RUNG
   RUNG wire#w1
      S_Coil( "UDT_Objetos".Valvulas."VM-39".control )
   END_RUNG
   RUNG wire#w1
      #TiempoEspera_Instance(Tiempo := "UDT_Objetos".Valvulas."VM-34".tiempo_alarma, Activacion := "UDT_Objetos".Valvulas."VM-39".control, Salida =>)
      Contact( #TiempoEspera_Instance.Salida )
      Contact( #PT073 )
      S_Coil( "UDT_Objetos".Bombas."BC-09".control )
   END_RUNG
   // the same network as SCL:
   IF #T4.Salida AND #RetrolavadoActivo AND NOT #RetrolavadoActivo2 THEN
       "UDT_Objetos".Valvulas."VM-34".control := TRUE;
       "UDT_Objetos".Valvulas."VM-39".control := TRUE;
   END_IF;
   #TiempoEspera_Instance(EN := #T4.Salida AND #RetrolavadoActivo AND NOT #RetrolavadoActivo2,   // "TiempoEspera"
                          Tiempo := "UDT_Objetos".Valvulas."VM-34".tiempo_alarma,
                          Activacion := "UDT_Objetos".Valvulas."VM-39".control,
                          ENO => #_w1);
   IF #_w1 AND #TiempoEspera_Instance.Salida AND #PT073 THEN
       "UDT_Objetos".Bombas."BC-09".control := TRUE;
   END_IF;
END_REGION

REGION Network 10: encendidoblower
   RUNG wire#powerrail
      Contact( #RetrolavadoActivo2 )
      I_Contact( #RetrolavadoActivo3 )
      #TiempoEspera_Instance_1(Tiempo := "UDT_Objetos".Valvulas."VM-39".tiempo_alarma, Activacion := #RetrolavadoActivo2, Salida =>)
      wire#w1
      R_Coil( "UDT_Objetos".Bombas."BC-09".control )
   END_RUNG
   RUNG wire#w1
      Contact( #TiempoEspera_Instance_1.Salida )
      R_Coil( "UDT_Objetos".Valvulas."VM-39".control )
   END_RUNG
   // the same network as SCL:
   #TiempoEspera_Instance_1(EN := #RetrolavadoActivo2 AND NOT #RetrolavadoActivo3,   // "TiempoEspera"
                           Tiempo := "UDT_Objetos".Valvulas."VM-39".tiempo_alarma,
                           Activacion := #RetrolavadoActivo2,
                           ENO => #_w1);
   IF #_w1 THEN "UDT_Objetos".Bombas."BC-09".control := FALSE; END_IF;
   IF #_w1 AND #TiempoEspera_Instance_1.Salida THEN "UDT_Objetos".Valvulas."VM-39".control := FALSE; END_IF;
END_REGION

REGION Network 11: activacion blower
   // ENO of a box is taken as its EN; it also drops when the box reports an error
   IF #RetrolavadoActivo AND #RetrolavadoActivo2 THEN
       #R_TRIG_Instance_1(CLK := "UDT_Objetos".Valvulas."VM-39".feedback);   // R_TRIG
   END_IF;
   #TiempoEspera_Instance_4(EN := #RetrolavadoActivo AND #RetrolavadoActivo2,   // "TiempoEspera"
                           Activacion := #R_TRIG_Instance_1.Q OR #F_TRIG_Instance.Q,
                           ENO => #_w1);
   IF #_w1 THEN "UDT_Objetos".Valvulas."VM-32".control := TRUE; END_IF;
   IF #_w1 AND #TiempoEspera_Instance_4.Salida THEN
       "UDT_Objetos".Equipos_Especiales."BLW-01".control := TRUE;
   END_IF;
   #_w2 := #RetrolavadoActivo AND #RetrolavadoActivo2;
   IF #_w2 THEN
       #F_TRIG_Instance(CLK := "UDT_Objetos".Valvulas."VM-39".feedback);   // F_TRIG
       #R_TRIG_Instance_2(CLK := #IEC_Timer_0_Instance_1.Q);   // R_TRIG
   END_IF;
   IF #_w2 AND #R_TRIG_Instance_2.Q THEN "UDT_Objetos".Valvulas."VM-33".control := TRUE; END_IF;
   #TiempoEspera_Instance_3(EN := #_w2,   // "TiempoEspera"
                           Tiempo := "UDT_Objetos".Valvulas."VM-32".tiempo_alarma,
                           Activacion := "UDT_Objetos".Valvulas."VM-33".control,
                           ENO => #_w3);
   IF #_w3 THEN "UDT_Objetos".Valvulas."VM-32".control := FALSE; END_IF;
   IF #_w3 AND #TiempoEspera_Instance_3.Salida THEN
       "UDT_Objetos".Equipos_Especiales."BLW-01".control := FALSE;
   END_IF;
END_REGION

REGION Network 12: apagar blower y tiempo valvula vm33
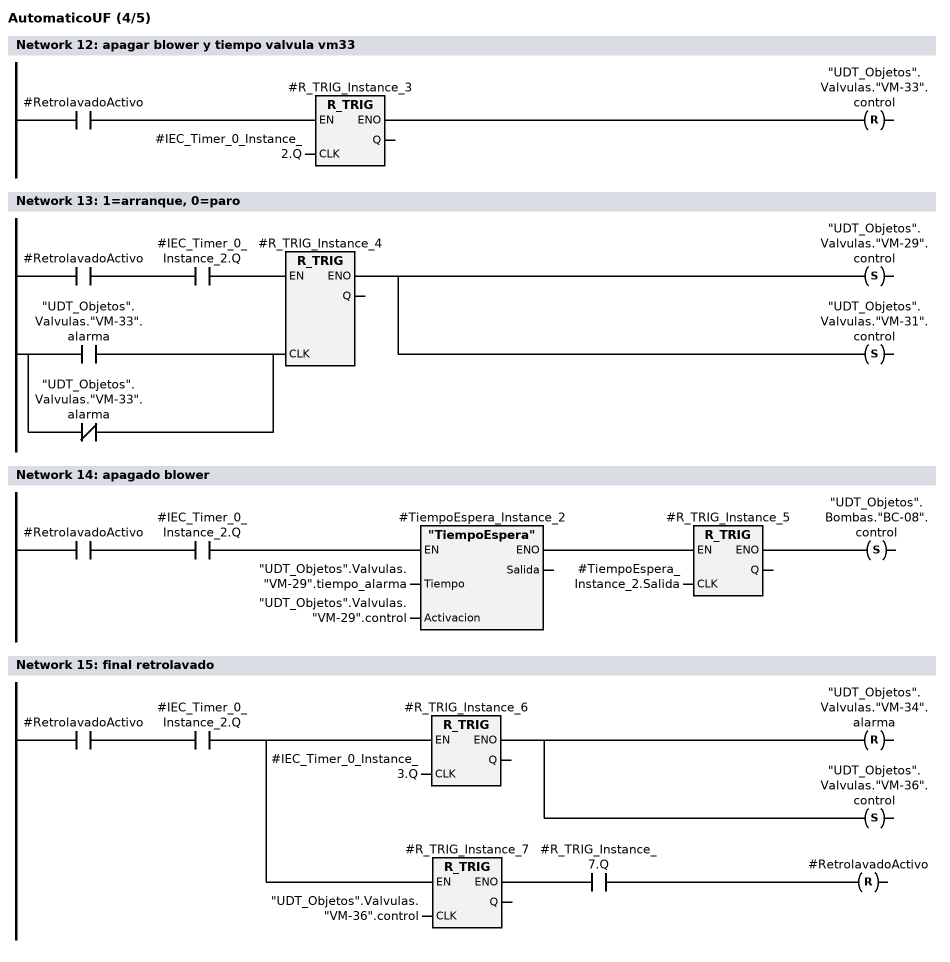
   // ENO of a box is taken as its EN; it also drops when the box reports an error
   IF #RetrolavadoActivo THEN
       #R_TRIG_Instance_3(CLK := #IEC_Timer_0_Instance_2.Q);   // R_TRIG
       "UDT_Objetos".Valvulas."VM-33".control := FALSE;
   END_IF;
END_REGION

REGION Network 13: 1=arranque, 0=paro
   // ENO of a box is taken as its EN; it also drops when the box reports an error
   IF #RetrolavadoActivo AND #IEC_Timer_0_Instance_2.Q THEN
       #R_TRIG_Instance_4(CLK := "UDT_Objetos".Valvulas."VM-33".alarma OR NOT "UDT_Objetos".Valvulas."VM-33".alarma);   // R_TRIG
       "UDT_Objetos".Valvulas."VM-29".control := TRUE;
       "UDT_Objetos".Valvulas."VM-31".control := TRUE;
   END_IF;
END_REGION

REGION Network 14: apagado blower
   // ENO of a box is taken as its EN; it also drops when the box reports an error
   #TiempoEspera_Instance_2(EN := #RetrolavadoActivo AND #IEC_Timer_0_Instance_2.Q,   // "TiempoEspera"
                           Tiempo := "UDT_Objetos".Valvulas."VM-29".tiempo_alarma,
                           Activacion := "UDT_Objetos".Valvulas."VM-29".control,
                           ENO => #_w1);
   IF #_w1 THEN
       #R_TRIG_Instance_5(CLK := #TiempoEspera_Instance_2.Salida);   // R_TRIG
       "UDT_Objetos".Bombas."BC-08".control := TRUE;
   END_IF;
END_REGION

REGION Network 15: final retrolavado
   // ENO of a box is taken as its EN; it also drops when the box reports an error
   #_w1 := #RetrolavadoActivo AND #IEC_Timer_0_Instance_2.Q;
   IF #_w1 THEN
       #R_TRIG_Instance_6(CLK := #IEC_Timer_0_Instance_3.Q);   // R_TRIG
       "UDT_Objetos".Valvulas."VM-34".alarma := FALSE;
       "UDT_Objetos".Valvulas."VM-36".control := TRUE;
       #R_TRIG_Instance_7(CLK := "UDT_Objetos".Valvulas."VM-36".control);   // R_TRIG
   END_IF;
   IF #_w1 AND #R_TRIG_Instance_7.Q THEN #RetrolavadoActivo := FALSE; END_IF;
END_REGION

REGION Network 16: BC-09 Y BC-10
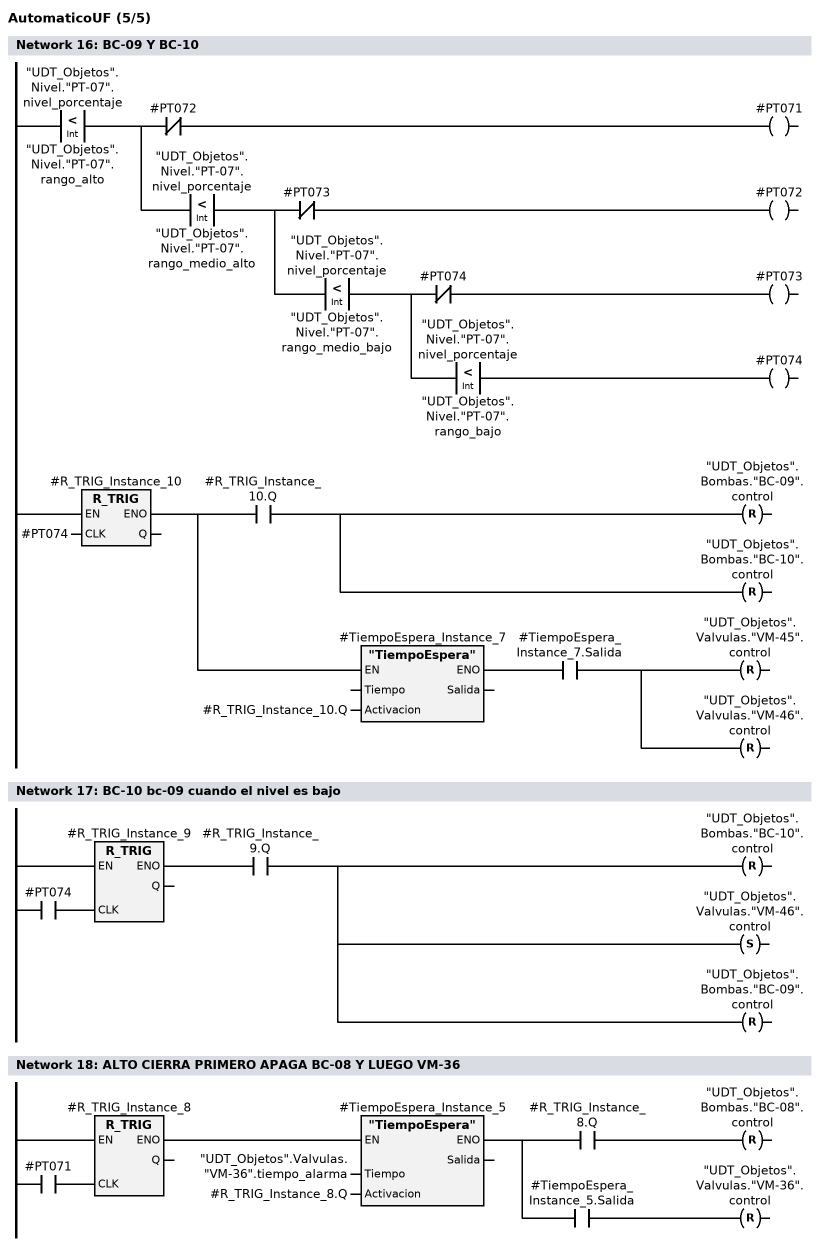
   // ENO of a box is taken as its EN; it also drops when the box reports an error
   #_w1 := "UDT_Objetos".Nivel."PT-07".nivel_porcentaje < "UDT_Objetos".Nivel."PT-07".rango_alto;
   #PT071 := #_w1 AND NOT #PT072;
   #_w2 := #_w1 AND ("UDT_Objetos".Nivel."PT-07".nivel_porcentaje < "UDT_Objetos".Nivel."PT-07".rango_medio_alto);
   #PT072 := #_w2 AND NOT #PT073;
   #_w3 := #_w2 AND ("UDT_Objetos".Nivel."PT-07".nivel_porcentaje < "UDT_Objetos".Nivel."PT-07".rango_medio_bajo);
   #PT073 := #_w3 AND NOT #PT074;
   #PT074 := #_w3 AND ("UDT_Objetos".Nivel."PT-07".nivel_porcentaje < "UDT_Objetos".Nivel."PT-07".rango_bajo);
   #R_TRIG_Instance_10(CLK := #PT074);   // R_TRIG
   IF #R_TRIG_Instance_10.Q THEN
       "UDT_Objetos".Bombas."BC-09".control := FALSE;
       "UDT_Objetos".Bombas."BC-10".control := FALSE;
   END_IF;
   #TiempoEspera_Instance_7(Activacion := #R_TRIG_Instance_10.Q, ENO => #_w4);   // "TiempoEspera"
   IF #_w4 AND #TiempoEspera_Instance_7.Salida THEN
       "UDT_Objetos".Valvulas."VM-45".control := FALSE;
       "UDT_Objetos".Valvulas."VM-46".control := FALSE;
   END_IF;
END_REGION

REGION Network 17: BC-10 bc-09 cuando el nivel es bajo
   // ENO of a box is taken as its EN; it also drops when the box reports an error
   #R_TRIG_Instance_9(CLK := #PT074);   // R_TRIG
   IF #R_TRIG_Instance_9.Q THEN
       "UDT_Objetos".Bombas."BC-10".control := FALSE;
       "UDT_Objetos".Valvulas."VM-46".control := TRUE;
       "UDT_Objetos".Bombas."BC-09".control := FALSE;
   END_IF;
END_REGION

REGION Network 18: ALTO CIERRA PRIMERO APAGA BC-08 Y LUEGO VM-36
   // ENO of a box is taken as its EN; it also drops when the box reports an error
   #R_TRIG_Instance_8(CLK := #PT071);   // R_TRIG
   #TiempoEspera_Instance_5(Tiempo := "UDT_Objetos".Valvulas."VM-36".tiempo_alarma,   // "TiempoEspera"
                           Activacion := #R_TRIG_Instance_8.Q,
                           ENO => #_w1);
   IF #_w1 AND #R_TRIG_Instance_8.Q THEN "UDT_Objetos".Bombas."BC-08".control := FALSE; END_IF;
   IF #_w1 AND #TiempoEspera_Instance_5.Salida THEN "UDT_Objetos".Valvulas."VM-36".control := FALSE; END_IF;
END_REGION
END_FUNCTION_BLOCK

FUNCTION_BLOCK "TiempoEspera"   // FB17, LAD
{ S7_Optimized_Access := 'TRUE' }
VERSION : 0.1
   VAR_INPUT
      Tiempo : Time;
      Activacion : Bool;
   END_VAR
   VAR_OUTPUT
      Salida : Bool;
   END_VAR
   VAR
      TP1 : TP_TIME;
      M1 : Bool;
   END_VAR
   VAR_TEMP
      Verdadero : Bool;
   END_VAR
   VAR_TEMP   // added for the SCL form of the ladder/FBD networks
      _w1 : Bool;
   END_VAR
BEGIN

REGION Network 1
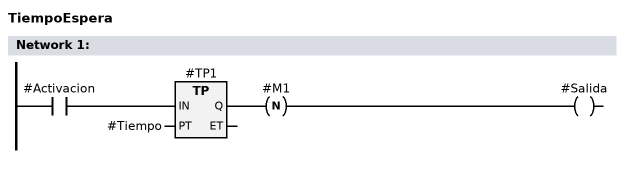
   #TP1(IN := #Activacion, PT := #Tiempo);   // TP
   #_w1 := NOT #TP1.Q AND #M1;   // falling edge
   #M1 := #TP1.Q;
   #Salida := #_w1;
END_REGION
END_FUNCTION_BLOCK

FUNCTION_BLOCK "AutomaticoOI"   // FB19, LAD
{ S7_Optimized_Access := 'TRUE' }
VERSION : 0.1
   VAR
      TiempoEspera_Instance_1 : "TiempoEspera";
      TiempoEspera_Instance_2 : "TiempoEspera";
   END_VAR
   VAR_TEMP   // added for the SCL form of the ladder/FBD networks
      _w1 : Bool;
      _w2 : Bool;
   END_VAR
BEGIN

REGION Network 1: ORP-01 Descarga bomba BC-10
END_REGION

REGION Network 2: ORP-01 Descarga bomba BC-10 SUPERIOR
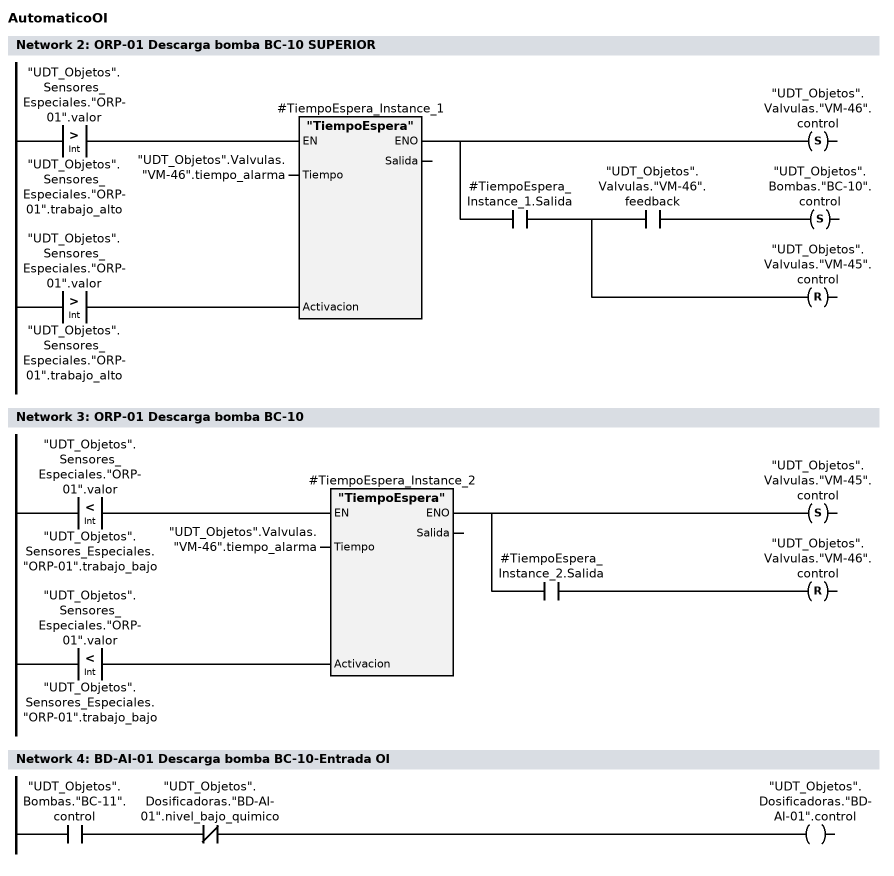
   RUNG wire#powerrail
      { S7_Templates := "SrcType := Int" } GT_Contact(in1 := "UDT_Objetos".Sensores_Especiales."ORP-01".valor, in2 := "UDT_Objetos".Sensores_Especiales."ORP-01".trabajo_alto)
      #TiempoEspera_Instance_1(Activacion := wire#w1, Tiempo := "UDT_Objetos".Valvulas."VM-46".tiempo_alarma, Salida =>)
      wire#w2
      S_Coil( "UDT_Objetos".Valvulas."VM-46".control )
   END_RUNG
   RUNG wire#powerrail
      { S7_Templates := "SrcType := Int" } GT_Contact(in1 := "UDT_Objetos".Sensores_Especiales."ORP-01".valor, in2 := "UDT_Objetos".Sensores_Especiales."ORP-01".trabajo_alto)
   END_RUNG wire#w1
   RUNG wire#w2
      Contact( #TiempoEspera_Instance_1.Salida )
      wire#w3
      Contact( "UDT_Objetos".Valvulas."VM-46".feedback )
      S_Coil( "UDT_Objetos".Bombas."BC-10".control )
   END_RUNG
   RUNG wire#w3
      R_Coil( "UDT_Objetos".Valvulas."VM-45".control )
   END_RUNG
   // the same network as SCL:
   #TiempoEspera_Instance_1(EN := "UDT_Objetos".Sensores_Especiales."ORP-01".valor > "UDT_Objetos".Sensores_Especiales."ORP-01".trabajo_alto,   // "TiempoEspera"
                           Tiempo := "UDT_Objetos".Valvulas."VM-46".tiempo_alarma,
                           Activacion := "UDT_Objetos".Sensores_Especiales."ORP-01".valor > "UDT_Objetos".Sensores_Especiales."ORP-01".trabajo_alto,
                           ENO => #_w1);
   IF #_w1 THEN "UDT_Objetos".Valvulas."VM-46".control := TRUE; END_IF;
   #_w2 := #_w1 AND #TiempoEspera_Instance_1.Salida;
   IF #_w2 AND "UDT_Objetos".Valvulas."VM-46".feedback THEN
       "UDT_Objetos".Bombas."BC-10".control := TRUE;
   END_IF;
   IF #_w2 THEN "UDT_Objetos".Valvulas."VM-45".control := FALSE; END_IF;
END_REGION

REGION Network 3: ORP-01 Descarga bomba BC-10
   RUNG wire#powerrail
      { S7_Templates := "SrcType := Int" } LT_Contact(in1 := "UDT_Objetos".Sensores_Especiales."ORP-01".valor, in2 := "UDT_Objetos".Sensores_Especiales."ORP-01".trabajo_bajo)
      #TiempoEspera_Instance_2(Activacion := wire#w1, Tiempo := "UDT_Objetos".Valvulas."VM-46".tiempo_alarma, Salida =>)
      wire#w2
      S_Coil( "UDT_Objetos".Valvulas."VM-45".control )
   END_RUNG
   RUNG wire#powerrail
      { S7_Templates := "SrcType := Int" } LT_Contact(in1 := "UDT_Objetos".Sensores_Especiales."ORP-01".valor, in2 := "UDT_Objetos".Sensores_Especiales."ORP-01".trabajo_bajo)
   END_RUNG wire#w1
   RUNG wire#w2
      Contact( #TiempoEspera_Instance_2.Salida )
      R_Coil( "UDT_Objetos".Valvulas."VM-46".control )
   END_RUNG
   // the same network as SCL:
   #TiempoEspera_Instance_2(EN := "UDT_Objetos".Sensores_Especiales."ORP-01".valor < "UDT_Objetos".Sensores_Especiales."ORP-01".trabajo_bajo,   // "TiempoEspera"
                           Tiempo := "UDT_Objetos".Valvulas."VM-46".tiempo_alarma,
                           Activacion := "UDT_Objetos".Sensores_Especiales."ORP-01".valor < "UDT_Objetos".Sensores_Especiales."ORP-01".trabajo_bajo,
                           ENO => #_w1);
   IF #_w1 THEN "UDT_Objetos".Valvulas."VM-45".control := TRUE; END_IF;
   IF #_w1 AND #TiempoEspera_Instance_2.Salida THEN "UDT_Objetos".Valvulas."VM-46".control := FALSE; END_IF;
END_REGION

REGION Network 4: BD-AI-01 Descarga bomba BC-10-Entrada OI
   RUNG wire#powerrail
      Contact( "UDT_Objetos".Bombas."BC-11".control )
      I_Contact( "UDT_Objetos".Dosificadoras."BD-AI-01".nivel_bajo_quimico )
      Coil( "UDT_Objetos".Dosificadoras."BD-AI-01".control )
   END_RUNG
   // the same network as SCL:
   "UDT_Objetos".Dosificadoras."BD-AI-01".control := "UDT_Objetos".Bombas."BC-11".control AND NOT "UDT_Objetos".Dosificadoras."BD-AI-01".nivel_bajo_quimico;
END_REGION

REGION Network 5: PT-09 Descarga bomba BC-11-OI
END_REGION
END_FUNCTION_BLOCK

ORGANIZATION_BLOCK "ProcesosMain"   // OB126, LAD, ProgramCycle
TITLE = "Main Program Sweep (Cycle)"
{ S7_Optimized_Access := 'TRUE' }
VERSION : 0.1
   VAR_INPUT
      Initial_Call : Bool;   // Initial call of this OB
      Remanence : Bool;   // =True, if remanent data are available
   END_VAR
BEGIN

REGION Network 1
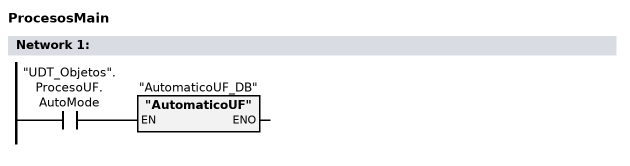
   RUNG wire#powerrail
      Contact( "UDT_Objetos".ProcesoUF.AutoMode )
      "AutomaticoUF_DB"()
   END_RUNG
   // the same network as SCL:
   IF "UDT_Objetos".ProcesoUF.AutoMode THEN
       "AutomaticoUF_DB"();   // "AutomaticoUF"
   END_IF;
END_REGION
END_ORGANIZATION_BLOCK

// folder: Transiciones_Entradas

FUNCTION "Escalizador_BC11" : Void   // FC2, LAD
{ S7_Optimized_Access := 'TRUE' }
VERSION : 0.1
   VAR_IN_OUT
      Bomba : "UDT_BOMBAS";
   END_VAR
   VAR_TEMP
      OutNormX : Real;
   END_VAR
BEGIN

REGION Network 1
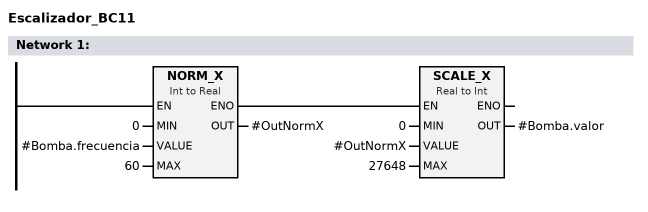
   RUNG wire#powerrail
      { S7_Templates := "[SrcType := Int, DestType := Real]"; S7_GenerateENO := "TRUE" } Normalize(min := 0, value := #Bomba.frecuencia, max := 60, out => #OutNormX)
      { S7_Templates := "[SrcType := Real, DestType := Int]"; S7_GenerateENO := "TRUE" } Scale(min := 0, value := #OutNormX, max := 27648, out => #Bomba.valor)
   END_RUNG
   // the same network as SCL:
   // ENO of a box is taken as its EN; it also drops when the box reports an error
   #OutNormX := NORM_X(MIN := 0, VALUE := #Bomba.frecuencia, MAX := 60);
   #Bomba.valor := SCALE_X(MIN := 0, VALUE := #OutNormX, MAX := 27648);
END_REGION
END_FUNCTION

FUNCTION "Nivel_PT_Escalizador" : Void   // FC3, LAD
{ S7_Optimized_Access := 'TRUE' }
VERSION : 0.1
   VAR_IN_OUT
      PT : "UDT_SENSORES_NIVEL";
   END_VAR
   VAR_TEMP
      OutNormX : Real;
      out : Real;
      Resultado_Transicion : Real;
      NiveAlto : Int;
      Resultado1 : Int;
      ResultadoNivel : Real;
      Escalizado : Real;
      M1 : Real;
   END_VAR
BEGIN

REGION Network 1
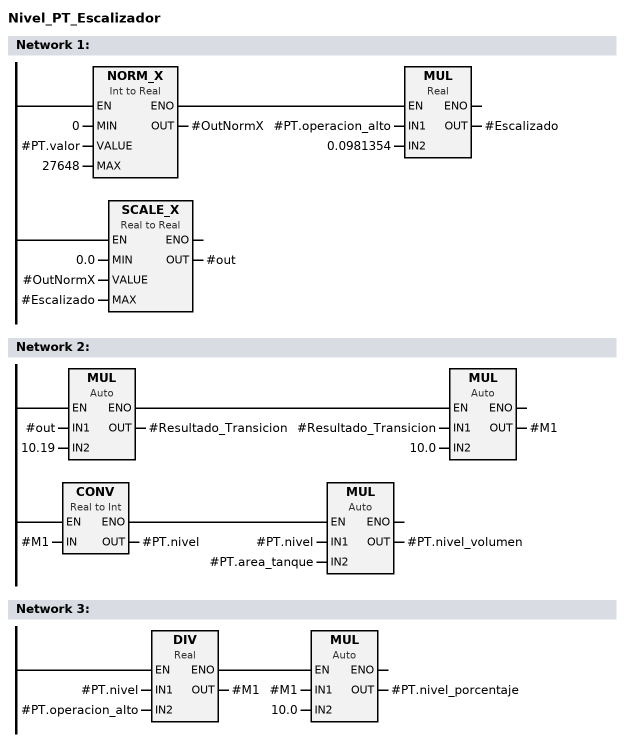
   RUNG wire#powerrail
      { S7_Templates := "[SrcType := Int, DestType := Real]"; S7_GenerateENO := "TRUE" } Normalize(min := 0, value := #PT.valor, max := 27648, out => #OutNormX)
      { S7_Templates := "SrcType := Real" } Mul(in1 := #PT.operacion_alto, in2 := 0.0981354, out => #Escalizado)
   END_RUNG
   RUNG wire#powerrail
      { S7_Templates := "[SrcType := Real, DestType := Real]"; S7_GenerateENO := "TRUE" } Scale(min := 0.0, value := #OutNormX, max := #Escalizado, out => #out)
   END_RUNG
   // the same network as SCL:
   // ENO of a box is taken as its EN; it also drops when the box reports an error
   #OutNormX := NORM_X(MIN := 0, VALUE := #PT.valor, MAX := 27648);
   #Escalizado := #PT.operacion_alto * 0.0981354;
   #out := SCALE_X(MIN := 0.0, VALUE := #OutNormX, MAX := #Escalizado);
END_REGION

REGION Network 2
   RUNG wire#powerrail
      Mul(in1 := #out, in2 := 10.19, out => #Resultado_Transicion)
      Mul(in1 := #Resultado_Transicion, in2 := 10.0, out => #M1)
   END_RUNG
   RUNG wire#powerrail
      { S7_Templates := "[SrcType := Real, DestType := Int]" } Convert(in := #M1, out => #PT.nivel)
      Mul(in1 := #PT.nivel, in2 := #PT.area_tanque, out => #PT.nivel_volumen)
   END_RUNG
   // the same network as SCL:
   #Resultado_Transicion := #out * 10.19;
   #M1 := #Resultado_Transicion * 10.0;
   #PT.nivel := REAL_TO_INT(#M1);
   #PT.nivel_volumen := #PT.nivel * #PT.area_tanque;
END_REGION

REGION Network 3
   RUNG wire#powerrail
      { S7_Templates := "SrcType := Real" } Div(in1 := #PT.nivel, in2 := #PT.operacion_alto, out => #M1)
      Mul(in1 := #M1, in2 := 10.0, out => #PT.nivel_porcentaje)
   END_RUNG
   // the same network as SCL:
   #M1 := #PT.nivel / #PT.operacion_alto;
   #PT.nivel_porcentaje := #M1 * 10.0;
END_REGION
END_FUNCTION

FUNCTION "Especiales_Escalizador" : Void   // FC4, LAD
{ S7_Optimized_Access := 'TRUE' }
VERSION : 0.1
   VAR_IN_OUT
      Especial : "UDT_SENSORES_ESPECIALES";
   END_VAR
   VAR_TEMP
      OutNormX : Real;
   END_VAR
BEGIN

REGION Network 1
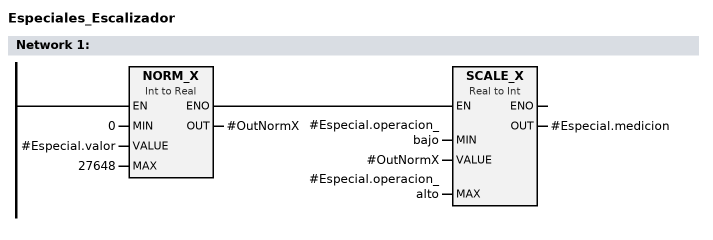
   RUNG wire#powerrail
      { S7_Templates := "[SrcType := Int, DestType := Real]"; S7_GenerateENO := "TRUE" } Normalize(min := 0, value := #Especial.valor, max := 27648, out => #OutNormX)
      { S7_Templates := "[SrcType := Real, DestType := Int]"; S7_GenerateENO := "TRUE" } Scale(min := #Especial.operacion_bajo, value := #OutNormX, max := #Especial.operacion_alto, out => #Especial.medicion)
   END_RUNG
   // the same network as SCL:
   // ENO of a box is taken as its EN; it also drops when the box reports an error
   #OutNormX := NORM_X(MIN := 0, VALUE := #Especial.valor, MAX := 27648);
   #Especial.medicion := SCALE_X(MIN := #Especial.operacion_bajo, VALUE := #OutNormX, MAX := #Especial.operacion_alto);
END_REGION
END_FUNCTION

FUNCTION "Presion_Escalizador" : Void   // FC5, LAD
{ S7_Optimized_Access := 'TRUE' }
VERSION : 0.1
   VAR_IN_OUT
      PT : "UDT_SENSORES_PRESION";
   END_VAR
   VAR_TEMP
      OutNormX : Real;
      out : Int;
      Resultado_Transicion : Int;
   END_VAR
BEGIN

REGION Network 1
